LIN {X 0,Y 227.871,Z 414.724,A -85,B 0,C 180,E1 -20018.086,E2 -20018.086} C_VEL
LIN {X 0,Y 228.23,Z 417.25,A -85,B 0,C 180,E1 -20022.645,E2 -20022.645} C_VEL
LIN {X 0,Y 228.444,Z 418.737,A -85,B 0,C 180,E1 -20025.039,E2 -20025.039} C_VEL
LIN {X 0,Y 228.671,Z 421.522,A -85,B 0,C 180,E1 -20029.238,E2 -20029.238} C_VEL
LIN {X 0,Y 228.672,Z 421.631,A -85,B 0,C 180,E1 -20029.384,E2 -20029.384} C_VEL
LIN {X 0,Y 229.708,Z 424.715,A -85,B 0,C 180,E1 -20029.753,E2 -20029.753} C_VEL
LIN {X 0,Y 231.122,Z 427.161,A -85,B 0,C 180,E1 -20030.178,E2 -20030.178} C_VEL
LIN {X 0,Y 235.965,Z 438.096,A -85,B 0,C 180,E1 -20031.887,E2 -20031.887} C_VEL
LIN {X 0,Y 239.913,Z 449.78,A -85,B 0,C 180,E1 -20033.668,E2 -20033.668} C_VEL
LIN {X 0,Y 243.067,Z 462.472,A -85,B 0,C 180,E1 -20035.659,E2 -20035.659} C_VEL
LIN {X 0,Y 244.778,Z 473.661,A -85,B 0,C 180,E1 -20037.501,E2 -20037.501} C_VEL
LIN {X 0,Y 245.596,Z 484.037,A -85,B 0,C 180,E1 -20039.347,E2 -20039.347} C_VEL
LIN {X 0,Y 242.616,Z 495.451,A -85,B 0,C 180,E1 -20041.211,E2 -20041.211} C_VEL
LIN {X 0,Y 239.291,Z 506.287,A -85,B 0,C 180,E1 -20043.392,E2 -20043.392} C_VEL
LIN {X 0,Y 236.26,Z 516.038,A -85,B 0,C 180,E1 -20045.857,E2 -20045.857} C_VEL
LIN {X 0,Y 233.502,Z 524.128,A -85,B 0,C 180,E1 -20048.364,E2 -20048.364} C_VEL
LIN {X 0,Y 231.017,Z 531.87,A -85,B 0,C 180,E1 -20051.372,E2 -20051.372} C_VEL
LIN {X 0,Y 229.237,Z 537.277,A -85,B 0,C 180,E1 -20053.983,E2 -20053.983} C_VEL
LIN {X 0,Y 227.771,Z 541.724,A -85,B 0,C 180,E1 -20056.62,E2 -20056.62} C_VEL
LIN {X 0,Y 226.783,Z 545.213,A -85,B 0,C 180,E1 -20059.284,E2 -20059.284} C_VEL
LIN {X 0,Y 226,Z 548.612,A -85,B 0,C 180,E1 -20062.855,E2 -20062.855} C_VEL
LIN {X 0,Y 225.629,Z 550.629,A -85,B 0,C 180,E1 -20066.428,E2 -20066.428} C_VEL
LIN {X 0,Y 225.637,Z 551.315,A -85,B 0,C 180,E1 -20070,E2 -20070} C_VEL
LIN {X 0,Y 225.629,Z 550.682,A -85,B 0,C 180,E1 -20073.572,E2 -20073.572} C_VEL
LIN {X 0,Y 225.998,Z 548.713,A -85,B 0,C 180,E1 -20077.146,E2 -20077.146} C_VEL
LIN {X 0,Y 226.763,Z 545.363,A -85,B 0,C 180,E1 -20080.717,E2 -20080.717} C_VEL
LIN {X 0,Y 228.133,Z 540.531,A -85,B 0,C 180,E1 -20084.268,E2 -20084.268} C_VEL
LIN {X 0,Y 230.402,Z 534.059,A -85,B 0,C 180,E1 -20087.76,E2 -20087.76} C_VEL
LIN {X 0,Y 232.445,Z 527.554,A -85,B 0,C 180,E1 -20090.519,E2 -20090.519} C_VEL
LIN {X 0,Y 235.212,Z 519.304,A -85,B 0,C 180,E1 -20093.323,E2 -20093.323} C_VEL
LIN {X 0,Y 238.194,Z 510.234,A -85,B 0,C 180,E1 -20095.799,E2 -20095.799} C_VEL
LIN {X 0,Y 241.6,Z 499.245,A -85,B 0,C 180,E1 -20098.21,E2 -20098.21} C_VEL
LIN {X 0,Y 244.722,Z 487.841,A -85,B 0,C 180,E1 -20100.206,E2 -20100.206} C_VEL
LIN {X 0,Y 245.654,Z 482.869,A -85,B 0,C 180,E1 -20100.996,E2 -20100.996} C_VEL
LIN {X 0,Y 244.462,Z 470.906,A -85,B 0,C 180,E1 -20103.109,E2 -20103.109} C_VEL
LIN {X 0,Y 242.661,Z 460.374,A -85,B 0,C 180,E1 -20104.815,E2 -20104.815} C_VEL
LIN {X 0,Y 239.265,Z 447.447,A -85,B 0,C 180,E1 -20106.828,E2 -20106.828} C_VEL
LIN {X 0,Y 235.103,Z 435.976,A -85,B 0,C 180,E1 -20108.587,E2 -20108.587} C_VEL
LIN {X 0,Y 232.091,Z 429.289,A -85,B 0,C 180,E1 -20109.642,E2 -20109.642} C_VEL
LIN {X 0,Y 230.405,Z 425.764,A -85,B 0,C 180,E1 -20110.203,E2 -20110.203} C_VEL
LIN {X 0,Y 228.882,Z 422.633,A -85,B 0,C 180,E1 -20110.677,E2 -20110.677} C_VEL
LIN {X 0,Y 228.676,Z 421.578,A -85,B 0,C 180,E1 -20110.836,E2 -20110.836} C_VEL
LIN {X 0,Y 228.449,Z 418.795,A -85,B 0,C 180,E1 -20115.038,E2 -20115.038} C_VEL
LIN {X 0,Y 228.031,Z 415.991,A -85,B 0,C 180,E1 -20119.667,E2 -20119.667} C_VEL
LIN {X 0,Y 227.849,Z 414.733,A -85,B 0,C 180,E1 -20121.91,E2 -20121.91} C_VEL
LIN {X 0,Y 227.881,Z 414.724,A -85,B 0,C 180,E1 -20126.377,E2 -20126.377} C_VEL
LIN {X 0,Y 227.922,Z 414.716,A -85,B 0,C 180,E1 -20130.438,E2 -20130.438} C_VEL
LIN {X 0,Y 227.931,Z 414.719,A -85,B 0,C 180,E1 -20134.426,E2 -20134.426} C_VEL
LIN {X 0,Y 227.965,Z 414.714,A -85,B 0,C 180,E1 -20138.287,E2 -20138.287} C_VEL
LIN {X 0,Y 228.037,Z 414.705,A -85,B 0,C 180,E1 -20142.825,E2 -20142.825} C_VEL
LIN {X 0,Y 228.097,Z 414.698,A -85,B 0,C 180,E1 -20147.544,E2 -20147.544} C_VEL
LIN {X 0,Y 228.328,Z 414.666,A -85,B 0,C 180,E1 -20151.147,E2 -20151.147} C_VEL
LIN {X 0,Y 228.361,Z 414.665,A -85,B 0,C 180,E1 -20152.929,E2 -20152.929} C_VEL
LIN {X 0,Y 228.557,Z 414.639,A -85,B 0,C 180,E1 -20158.238,E2 -20158.238} C_VEL
LIN {X 0,Y 228.558,Z 414.641,A -85,B 0,C 180,E1 -20161.762,E2 -20161.762} C_VEL
LIN {X 0,Y 228.361,Z 414.665,A -85,B 0,C 180,E1 -20167.071,E2 -20167.071} C_VEL
LIN {X 0,Y 228.174,Z 414.687,A -85,B 0,C 180,E1 -20170.65,E2 -20170.65} C_VEL
LIN {X 0,Y 228.06,Z 414.704,A -85,B 0,C 180,E1 -20176.102,E2 -20176.102} C_VEL
LIN {X 0,Y 227.945,Z 414.718,A -85,B 0,C 180,E1 -20179.825,E2 -20179.825} C_VEL
LIN {X 0,Y 227.916,Z 414.713,A -85,B 0,C 180,E1 -20183.632,E2 -20183.632} C_VEL
LIN {X 0,Y 227.888,Z 414.718,A -85,B 0,C 180,E1 -20187.555,E2 -20187.555} C_VEL
LIN {X 0,Y 227.875,Z 414.726,A -85,B 0,C 180,E1 -20191.621,E2 -20191.621} C_VEL
LIN {X 0,Y 227.892,Z 414.725,A -85,B 0,C 180,E1 -20193.718,E2 -20193.718} C_VEL
LIN {X 0,Y 228.131,Z 416.119,A -85,B 0,C 180,E1 -20196.776,E2 -20196.776} C_VEL
LIN {X 0,Y 228.439,Z 418.282,A -85,B 0,C 180,E1 -20200.246,E2 -20200.246} C_VEL
LIN {X 0,Y 228.732,Z 419.796,A -85,B 0,C 180,E1 -20202.53,E2 -20202.53} C_VEL
LIN {X 0,Y 228.948,Z 421.571,A -85,B 0,C 180,E1 -20205.087,E2 -20205.087} C_VEL
LIN {X 0,Y 229.149,Z 424.277,A -85,B 0,C 180,E1 -20208.712,E2 -20208.712} C_VEL
LIN {X 0,Y 229.127,Z 424.775,A -85,B 0,C 180,E1 -20209.344,E2 -20209.344} C_VEL
LIN {X 0,Y 230.212,Z 428.044,A -85,B 0,C 180,E1 -20209.748,E2 -20209.748} C_VEL
LIN {X 0,Y 231.469,Z 430.266,A -85,B 0,C 180,E1 -20210.122,E2 -20210.122} C_VEL
LIN {X 0,Y 235.394,Z 439.747,A -85,B 0,C 180,E1 -20211.529,E2 -20211.529} C_VEL
LIN {X 0,Y 239.443,Z 452.197,A -85,B 0,C 180,E1 -20213.352,E2 -20213.352} C_VEL
LIN {X 0,Y 240.173,Z 457.38,A -85,B 0,C 180,E1 -20214.014,E2 -20214.014} C_VEL
LIN {X 0,Y 239.976,Z 462.788,A -85,B 0,C 180,E1 -20214.601,E2 -20214.601} C_VEL
LIN {X 0,Y 238.366,Z 473.596,A -85,B 0,C 180,E1 -20215.801,E2 -20215.801} C_VEL
LIN {X 0,Y 237.926,Z 478.732,A -85,B 0,C 180,E1 -20216.526,E2 -20216.526} C_VEL
LIN {X 0,Y 237.969,Z 480.365,A -85,B 0,C 180,E1 -20216.8,E2 -20216.8} C_VEL
LIN {X 0,Y 238.435,Z 490.141,A -85,B 0,C 180,E1 -20218.626,E2 -20218.626} C_VEL
LIN {X 0,Y 235.967,Z 499.91,A -85,B 0,C 180,E1 -20220.32,E2 -20220.32} C_VEL
LIN {X 0,Y 232.489,Z 510.701,A -85,B 0,C 180,E1 -20222.548,E2 -20222.548} C_VEL
LIN {X 0,Y 229.263,Z 520.429,A -85,B 0,C 180,E1 -20225.07,E2 -20225.07} C_VEL
LIN {X 0,Y 226.424,Z 528.498,A -85,B 0,C 180,E1 -20227.652,E2 -20227.652} C_VEL
LIN {X 0,Y 224.105,Z 534.99,A -85,B 0,C 180,E1 -20230.187,E2 -20230.187} C_VEL
LIN {X 0,Y 222.033,Z 541.634,A -85,B 0,C 180,E1 -20233.448,E2 -20233.448} C_VEL
LIN {X 0,Y 220.123,Z 547.315,A -85,B 0,C 180,E1 -20237.085,E2 -20237.085} C_VEL
LIN {X 0,Y 219.076,Z 551.438,A -85,B 0,C 180,E1 -20240.77,E2 -20240.77} C_VEL
LIN {X 0,Y 218.567,Z 554.13,A -85,B 0,C 180,E1 -20244.464,E2 -20244.464} C_VEL
LIN {X 0,Y 218.467,Z 555.461,A -85,B 0,C 180,E1 -20248.156,E2 -20248.156} C_VEL
LIN {X 0,Y 218.532,Z 555.625,A -85,B 0,C 180,E1 -20250,E2 -20250} C_VEL
LIN {X 0,Y 218.449,Z 554.948,A -85,B 0,C 180,E1 -20253.689,E2 -20253.689} C_VEL
LIN {X 0,Y 218.758,Z 552.928,A -85,B 0,C 180,E1 -20257.383,E2 -20257.383} C_VEL
LIN {X 0,Y 219.552,Z 549.517,A -85,B 0,C 180,E1 -20261.073,E2 -20261.073} C_VEL
LIN {X 0,Y 220.952,Z 544.612,A -85,B 0,C 180,E1 -20264.742,E2 -20264.742} C_VEL
LIN {X 0,Y 222.567,Z 539.883,A -85,B 0,C 180,E1 -20267.456,E2 -20267.456} C_VEL
LIN {X 0,Y 224.851,Z 533.028,A -85,B 0,C 180,E1 -20270.587,E2 -20270.587} C_VEL
LIN {X 0,Y 227.79,Z 524.519,A -85,B 0,C 180,E1 -20273.646,E2 -20273.646} C_VEL
LIN {X 0,Y 230.836,Z 515.642,A -85,B 0,C 180,E1 -20276.197,E2 -20276.197} C_VEL
LIN {X 0,Y 234.347,Z 504.889,A -85,B 0,C 180,E1 -20278.675,E2 -20278.675} C_VEL
LIN {X 0,Y 237.768,Z 493.13,A -85,B 0,C 180,E1 -20280.839,E2 -20280.839} C_VEL
LIN {X 0,Y 238.393,Z 489.802,A -85,B 0,C 180,E1 -20281.396,E2 -20281.396} C_VEL
LIN {X 0,Y 237.762,Z 478.712,A -85,B 0,C 180,E1 -20283.448,E2 -20283.448} C_VEL
LIN {X 0,Y 236.133,Z 466.35,A -85,B 0,C 180,E1 -20285.536,E2 -20285.536} C_VEL
LIN {X 0,Y 233.476,Z 454.446,A -85,B 0,C 180,E1 -20287.445,E2 -20287.445} C_VEL
LIN {X 0,Y 229.625,Z 442.08,A -85,B 0,C 180,E1 -20289.376,E2 -20289.376} C_VEL
LIN {X 0,Y 226.084,Z 433.454,A -85,B 0,C 180,E1 -20290.753,E2 -20290.753} C_VEL
LIN {X 0,Y 223.799,Z 428.789,A -85,B 0,C 180,E1 -20291.548,E2 -20291.548} C_VEL
LIN {X 0,Y 222.268,Z 425.689,A -85,B 0,C 180,E1 -20292.054,E2 -20292.054} C_VEL
LIN {X 0,Y 222.084,Z 424.67,A -85,B 0,C 180,E1 -20292.188,E2 -20292.188} C_VEL
LIN {X 0,Y 221.733,Z 421.441,A -85,B 0,C 180,E1 -20296.803,E2 -20296.803} C_VEL
LIN {X 0,Y 221.37,Z 419.006,A -85,B 0,C 180,E1 -20300.583,E2 -20300.583} C_VEL
LIN {X 0,Y 220.945,Z 416.375,A -85,B 0,C 180,E1 -20305.071,E2 -20305.071} C_VEL
LIN {X 0,Y 220.824,Z 415.606,A -85,B 0,C 180,E1 -20307.245,E2 -20307.245} C_VEL
LIN {X 0,Y 220.827,Z 415.604,A -85,B 0,C 180,E1 -20311.485,E2 -20311.485} C_VEL
LIN {X 0,Y 220.863,Z 415.599,A -85,B 0,C 180,E1 -20315.565,E2 -20315.565} C_VEL
LIN {X 0,Y 220.886,Z 415.596,A -85,B 0,C 180,E1 -20319.513,E2 -20319.513} C_VEL
LIN {X 0,Y 221.018,Z 415.579,A -85,B 0,C 180,E1 -20323.37,E2 -20323.37} C_VEL
LIN {X 0,Y 221.118,Z 415.561,A -85,B 0,C 180,E1 -20329.006,E2 -20329.006} C_VEL
LIN {X 0,Y 221.313,Z 415.535,A -85,B 0,C 180,E1 -20332.702,E2 -20332.702} C_VEL
LIN {X 0,Y 221.515,Z 415.517,A -85,B 0,C 180,E1 -20338.182,E2 -20338.182} C_VEL
LIN {X 0,Y 221.514,Z 415.517,A -85,B 0,C 180,E1 -20341.818,E2 -20341.818} C_VEL
LIN {X 0,Y 221.313,Z 415.543,A -85,B 0,C 180,E1 -20347.298,E2 -20347.298} C_VEL
LIN {X 0,Y 221.118,Z 415.566,A -85,B 0,C 180,E1 -20350.994,E2 -20350.994} C_VEL
LIN {X 0,Y 221.018,Z 415.574,A -85,B 0,C 180,E1 -20356.63,E2 -20356.63} C_VEL
LIN {X 0,Y 220.894,Z 415.595,A -85,B 0,C 180,E1 -20360.486,E2 -20360.486} C_VEL
LIN {X 0,Y 220.869,Z 415.598,A -85,B 0,C 180,E1 -20364.435,E2 -20364.435} C_VEL
LIN {X 0,Y 220.828,Z 415.603,A -85,B 0,C 180,E1 -20368.515,E2 -20368.515} C_VEL
LIN {X 0,Y 220.824,Z 415.604,A -85,B 0,C 180,E1 -20372.755,E2 -20372.755} C_VEL
LIN {X 0,Y 220.839,Z 415.603,A -85,B 0,C 180,E1 -20377.288,E2 -20377.288} C_VEL
LIN {X 0,Y 221.18,Z 418.058,A -85,B 0,C 180,E1 -20381.857,E2 -20381.857} C_VEL
LIN {X 0,Y 221.472,Z 420.385,A -85,B 0,C 180,E1 -20385.723,E2 -20385.723} C_VEL
LIN {X 0,Y 221.635,Z 421.75,A -85,B 0,C 180,E1 -20387.805,E2 -20387.805} C_VEL
LIN {X 0,Y 222.739,Z 424.806,A -85,B 0,C 180,E1 -20388.217,E2 -20388.217} C_VEL
LIN {X 0,Y 224.207,Z 427.147,A -85,B 0,C 180,E1 -20388.68,E2 -20388.68} C_VEL
LIN {X 0,Y 229.392,Z 438.499,A -85,B 0,C 180,E1 -20390.611,E2 -20390.611} C_VEL
LIN {X 0,Y 233.08,Z 448.969,A -85,B 0,C 180,E1 -20392.328,E2 -20392.328} C_VEL
LIN {X 0,Y 236.412,Z 461.889,A -85,B 0,C 180,E1 -20394.462,E2 -20394.462} C_VEL
LIN {X 0,Y 238.314,Z 473.741,A -85,B 0,C 180,E1 -20396.505,E2 -20396.505} C_VEL
LIN {X 0,Y 239.179,Z 484.183,A -85,B 0,C 180,E1 -20398.445,E2 -20398.445} C_VEL
LIN {X 0,Y 238.474,Z 488.194,A -85,B 0,C 180,E1 -20399.11,E2 -20399.11} C_VEL
LIN {X 0,Y 235.433,Z 498.727,A -85,B 0,C 180,E1 -20400.982,E2 -20400.982} C_VEL
LIN {X 0,Y 232.395,Z 508.137,A -85,B 0,C 180,E1 -20403.024,E2 -20403.024} C_VEL
LIN {X 0,Y 229.244,Z 517.592,A -85,B 0,C 180,E1 -20405.552,E2 -20405.552} C_VEL
LIN {X 0,Y 226.026,Z 526.63,A -85,B 0,C 180,E1 -20408.58,E2 -20408.58} C_VEL
LIN {X 0,Y 223.66,Z 533.87,A -85,B 0,C 180,E1 -20411.686,E2 -20411.686} C_VEL
LIN {X 0,Y 221.248,Z 540.395,A -85,B 0,C 180,E1 -20415.279,E2 -20415.279} C_VEL
LIN {X 0,Y 219.772,Z 545.283,A -85,B 0,C 180,E1 -20418.938,E2 -20418.938} C_VEL
LIN {X 0,Y 218.943,Z 548.682,A -85,B 0,C 180,E1 -20422.623,E2 -20422.623} C_VEL
LIN {X 0,Y 218.534,Z 550.698,A -85,B 0,C 180,E1 -20426.312,E2 -20426.312} C_VEL
LIN {X 0,Y 218.537,Z 551.384,A -85,B 0,C 180,E1 -20430,E2 -20430} C_VEL
LIN {X 0,Y 218.534,Z 550.751,A -85,B 0,C 180,E1 -20433.688,E2 -20433.688} C_VEL
LIN {X 0,Y 218.941,Z 548.781,A -85,B 0,C 180,E1 -20437.377,E2 -20437.377} C_VEL
LIN {X 0,Y 219.75,Z 545.431,A -85,B 0,C 180,E1 -20441.063,E2 -20441.063} C_VEL
LIN {X 0,Y 221.225,Z 540.599,A -85,B 0,C 180,E1 -20444.723,E2 -20444.723} C_VEL
LIN {X 0,Y 222.978,Z 535.932,A -85,B 0,C 180,E1 -20447.423,E2 -20447.423} C_VEL
LIN {X 0,Y 225.301,Z 528.928,A -85,B 0,C 180,E1 -20450.639,E2 -20450.639} C_VEL
LIN {X 0,Y 228.203,Z 520.722,A -85,B 0,C 180,E1 -20453.601,E2 -20453.601} C_VEL
LIN {X 0,Y 231.227,Z 511.925,A -85,B 0,C 180,E1 -20456.15,E2 -20456.15} C_VEL
LIN {X 0,Y 234.73,Z 501.263,A -85,B 0,C 180,E1 -20458.624,E2 -20458.624} C_VEL
LIN {X 0,Y 238.108,Z 489.742,A -85,B 0,C 180,E1 -20460.762,E2 -20460.762} C_VEL
LIN {X 0,Y 239.256,Z 484.688,A -85,B 0,C 180,E1 -20461.585,E2 -20461.585} C_VEL
LIN {X 0,Y 238.265,Z 473.172,A -85,B 0,C 180,E1 -20463.735,E2 -20463.735} C_VEL
LIN {X 0,Y 236.669,Z 462.938,A -85,B 0,C 180,E1 -20465.5,E2 -20465.5} C_VEL
LIN {X 0,Y 233.693,Z 450.793,A -85,B 0,C 180,E1 -20467.514,E2 -20467.514} C_VEL
LIN {X 0,Y 229.547,Z 438.758,A -85,B 0,C 180,E1 -20469.491,E2 -20469.491} C_VEL
LIN {X 0,Y 225.551,Z 430.034,A -85,B 0,C 180,E1 -20470.988,E2 -20470.988} C_VEL
LIN {X 0,Y 223.627,Z 426.043,A -85,B 0,C 180,E1 -20471.676,E2 -20471.676} C_VEL
LIN {X 0,Y 222.021,Z 423.296,A -85,B 0,C 180,E1 -20472.186,E2 -20472.186} C_VEL
LIN {X 0,Y 221.616,Z 421.7,A -85,B 0,C 180,E1 -20472.386,E2 -20472.386} C_VEL
LIN {X 0,Y 221.263,Z 418.872,A -85,B 0,C 180,E1 -20476.933,E2 -20476.933} C_VEL
LIN {X 0,Y 221,Z 416.838,A -85,B 0,C 180,E1 -20480.504,E2 -20480.504} C_VEL
LIN {X 0,Y 220.826,Z 415.615,A -85,B 0,C 180,E1 -20482.793,E2 -20482.793} C_VEL
LIN {X 0,Y 220.82,Z 415.604,A -85,B 0,C 180,E1 -20487.244,E2 -20487.244} C_VEL
LIN {X 0,Y 220.839,Z 415.602,A -85,B 0,C 180,E1 -20491.487,E2 -20491.487} C_VEL
LIN {X 0,Y 220.87,Z 415.595,A -85,B 0,C 180,E1 -20495.565,E2 -20495.565} C_VEL
LIN {X 0,Y 220.895,Z 415.588,A -85,B 0,C 180,E1 -20499.514,E2 -20499.514} C_VEL
LIN {X 0,Y 221.019,Z 415.58,A -85,B 0,C 180,E1 -20503.37,E2 -20503.37} C_VEL
LIN {X 0,Y 221.12,Z 415.566,A -85,B 0,C 180,E1 -20509.006,E2 -20509.006} C_VEL
LIN {X 0,Y 221.314,Z 415.542,A -85,B 0,C 180,E1 -20512.702,E2 -20512.702} C_VEL
LIN {X 0,Y 221.515,Z 415.516,A -85,B 0,C 180,E1 -20518.182,E2 -20518.182} C_VEL
LIN {X 0,Y 221.516,Z 415.518,A -85,B 0,C 180,E1 -20521.818,E2 -20521.818} C_VEL
LIN {X 0,Y 221.314,Z 415.542,A -85,B 0,C 180,E1 -20527.297,E2 -20527.297} C_VEL
LIN {X 0,Y 221.119,Z 415.566,A -85,B 0,C 180,E1 -20530.994,E2 -20530.994} C_VEL
LIN {X 0,Y 221.019,Z 415.578,A -85,B 0,C 180,E1 -20536.629,E2 -20536.629} C_VEL
LIN {X 0,Y 220.895,Z 415.595,A -85,B 0,C 180,E1 -20540.486,E2 -20540.486} C_VEL
LIN {X 0,Y 220.869,Z 415.591,A -85,B 0,C 180,E1 -20544.435,E2 -20544.435} C_VEL
LIN {X 0,Y 220.839,Z 415.602,A -85,B 0,C 180,E1 -20548.513,E2 -20548.513} C_VEL
LIN {X 0,Y 220.826,Z 415.604,A -85,B 0,C 180,E1 -20552.754,E2 -20552.754} C_VEL
LIN {X 0,Y 220.954,Z 416.433,A -85,B 0,C 180,E1 -20554.927,E2 -20554.927} C_VEL
LIN {X 0,Y 221.378,Z 419.059,A -85,B 0,C 180,E1 -20559.415,E2 -20559.415} C_VEL
LIN {X 0,Y 221.756,Z 421.493,A -85,B 0,C 180,E1 -20563.203,E2 -20563.203} C_VEL
LIN {X 0,Y 222.158,Z 424.853,A -85,B 0,C 180,E1 -20567.808,E2 -20567.808} C_VEL
LIN {X 0,Y 223.3,Z 428.018,A -85,B 0,C 180,E1 -20568.231,E2 -20568.231} C_VEL
LIN {X 0,Y 224.65,Z 430.332,A -85,B 0,C 180,E1 -20568.661,E2 -20568.661} C_VEL
LIN {X 0,Y 229.373,Z 441.097,A -85,B 0,C 180,E1 -20570.434,E2 -20570.434} C_VEL
LIN {X 0,Y 233.591,Z 454.451,A -85,B 0,C 180,E1 -20572.519,E2 -20572.519} C_VEL
LIN {X 0,Y 235.977,Z 465.2,A -85,B 0,C 180,E1 -20574.231,E2 -20574.231} C_VEL
LIN {X 0,Y 237.489,Z 475.583,A -85,B 0,C 180,E1 -20575.956,E2 -20575.956} C_VEL
LIN {X 0,Y 237.969,Z 480.365,A -85,B 0,C 180,E1 -20576.8,E2 -20576.8} C_VEL
LIN {X 0,Y 237.788,Z 483.651,A -85,B 0,C 180,E1 -20577.331,E2 -20577.331} C_VEL
LIN {X 0,Y 236.364,Z 488.667,A -85,B 0,C 180,E1 -20578.031,E2 -20578.031} C_VEL
LIN {X 0,Y 234.087,Z 493.547,A -85,B 0,C 180,E1 -20578.67,E2 -20578.67} C_VEL
LIN {X 0,Y 229.005,Z 503.067,A -85,B 0,C 180,E1 -20580.09,E2 -20580.09} C_VEL
LIN {X 0,Y 227.778,Z 506.04,A -85,B 0,C 180,E1 -20580.685,E2 -20580.685} C_VEL
LIN {X 0,Y 224.427,Z 515.73,A -85,B 0,C 180,E1 -20582.995,E2 -20582.995} C_VEL
LIN {X 0,Y 221.297,Z 524.581,A -85,B 0,C 180,E1 -20585.615,E2 -20585.615} C_VEL
LIN {X 0,Y 218.145,Z 533.064,A -85,B 0,C 180,E1 -20588.749,E2 -20588.749} C_VEL
LIN {X 0,Y 215.743,Z 539.901,A -85,B 0,C 180,E1 -20591.972,E2 -20591.972} C_VEL
LIN {X 0,Y 214.077,Z 544.611,A -85,B 0,C 180,E1 -20594.773,E2 -20594.773} C_VEL
LIN {X 0,Y 212.546,Z 549.494,A -85,B 0,C 180,E1 -20598.557,E2 -20598.557} C_VEL
LIN {X 0,Y 211.667,Z 552.888,A -85,B 0,C 180,E1 -20602.368,E2 -20602.368} C_VEL
LIN {X 0,Y 211.349,Z 554.895,A -85,B 0,C 180,E1 -20606.186,E2 -20606.186} C_VEL
LIN {X 0,Y 211.434,Z 555.556,A -85,B 0,C 180,E1 -20610,E2 -20610} C_VEL
LIN {X 0,Y 211.354,Z 554.878,A -85,B 0,C 180,E1 -20613.813,E2 -20613.813} C_VEL
LIN {X 0,Y 211.685,Z 552.858,A -85,B 0,C 180,E1 -20617.631,E2 -20617.631} C_VEL
LIN {X 0,Y 212.534,Z 549.446,A -85,B 0,C 180,E1 -20621.444,E2 -20621.444} C_VEL
LIN {X 0,Y 214.075,Z 544.541,A -85,B 0,C 180,E1 -20625.226,E2 -20625.226} C_VEL
LIN {X 0,Y 216.442,Z 538,A -85,B 0,C 180,E1 -20628.948,E2 -20628.948} C_VEL
LIN {X 0,Y 218.959,Z 530.72,A -85,B 0,C 180,E1 -20632.157,E2 -20632.157} C_VEL
LIN {X 0,Y 222.296,Z 521.703,A -85,B 0,C 180,E1 -20635.265,E2 -20635.265} C_VEL
LIN {X 0,Y 225.578,Z 512.242,A -85,B 0,C 180,E1 -20637.861,E2 -20637.861} C_VEL
LIN {X 0,Y 229.095,Z 501.769,A -85,B 0,C 180,E1 -20640.155,E2 -20640.155} C_VEL
LIN {X 0,Y 231.991,Z 491.683,A -85,B 0,C 180,E1 -20641.979,E2 -20641.979} C_VEL
LIN {X 0,Y 231.584,Z 481.339,A -85,B 0,C 180,E1 -20644.008,E2 -20644.008} C_VEL
LIN {X 0,Y 230.147,Z 468.823,A -85,B 0,C 180,E1 -20646.257,E2 -20646.257} C_VEL
LIN {X 0,Y 227.602,Z 456.606,A -85,B 0,C 180,E1 -20648.335,E2 -20648.335} C_VEL
LIN {X 0,Y 223.683,Z 443.741,A -85,B 0,C 180,E1 -20650.484,E2 -20650.484} C_VEL
LIN {X 0,Y 219.427,Z 433.674,A -85,B 0,C 180,E1 -20652.246,E2 -20652.246} C_VEL
LIN {X 0,Y 217.641,Z 429.973,A -85,B 0,C 180,E1 -20652.928,E2 -20652.928} C_VEL
LIN {X 0,Y 215.472,Z 426.425,A -85,B 0,C 180,E1 -20653.661,E2 -20653.661} C_VEL
LIN {X 0,Y 214.984,Z 424.57,A -85,B 0,C 180,E1 -20653.951,E2 -20653.951} C_VEL
LIN {X 0,Y 214.756,Z 422.805,A -85,B 0,C 180,E1 -20656.588,E2 -20656.588} C_VEL
LIN {X 0,Y 214.538,Z 421.232,A -85,B 0,C 180,E1 -20659.067,E2 -20659.067} C_VEL
LIN {X 0,Y 214.081,Z 418.468,A -85,B 0,C 180,E1 -20663.778,E2 -20663.778} C_VEL
LIN {X 0,Y 213.903,Z 417.245,A -85,B 0,C 180,E1 -20666.044,E2 -20666.044} C_VEL
LIN {X 0,Y 213.782,Z 416.484,A -85,B 0,C 180,E1 -20668.731,E2 -20668.731} C_VEL
LIN {X 0,Y 213.827,Z 416.476,A -85,B 0,C 180,E1 -20672.603,E2 -20672.603} C_VEL
LIN {X 0,Y 213.82,Z 416.476,A -85,B 0,C 180,E1 -20676.974,E2 -20676.974} C_VEL
LIN {X 0,Y 213.945,Z 416.457,A -85,B 0,C 180,E1 -20682.804,E2 -20682.804} C_VEL
LIN {X 0,Y 213.982,Z 416.455,A -85,B 0,C 180,E1 -20686.709,E2 -20686.709} C_VEL
LIN {X 0,Y 214.198,Z 416.43,A -85,B 0,C 180,E1 -20690.558,E2 -20690.558} C_VEL
LIN {X 0,Y 214.25,Z 416.415,A -85,B 0,C 180,E1 -20692.461,E2 -20692.461} C_VEL
LIN {X 0,Y 214.448,Z 416.397,A -85,B 0,C 180,E1 -20698.122,E2 -20698.122} C_VEL
LIN {X 0,Y 214.556,Z 416.383,A -85,B 0,C 180,E1 -20700,E2 -20700} C_VEL
LIN {X 0,Y 214.447,Z 416.397,A -85,B 0,C 180,E1 -20701.878,E2 -20701.878} C_VEL
LIN {X 0,Y 214.25,Z 416.423,A -85,B 0,C 180,E1 -20707.54,E2 -20707.54} C_VEL
LIN {X 0,Y 214.049,Z 416.448,A -85,B 0,C 180,E1 -20711.362,E2 -20711.362} C_VEL
LIN {X 0,Y 213.936,Z 416.462,A -85,B 0,C 180,E1 -20715.237,E2 -20715.237} C_VEL
LIN {X 0,Y 213.842,Z 416.474,A -85,B 0,C 180,E1 -20719.187,E2 -20719.187} C_VEL
LIN {X 0,Y 213.849,Z 416.472,A -85,B 0,C 180,E1 -20723.227,E2 -20723.227} C_VEL
LIN {X 0,Y 213.83,Z 416.474,A -85,B 0,C 180,E1 -20727.45,E2 -20727.45} C_VEL
LIN {X 0,Y 213.771,Z 416.483,A -85,B 0,C 180,E1 -20731.737,E2 -20731.737} C_VEL
LIN {X 0,Y 213.754,Z 416.486,A -85,B 0,C 180,E1 -20736.287,E2 -20736.287} C_VEL
LIN {X 0,Y 214.126,Z 418.891,A -85,B 0,C 180,E1 -20741.029,E2 -20741.029} C_VEL
LIN {X 0,Y 214.488,Z 421.794,A -85,B 0,C 180,E1 -20746.045,E2 -20746.045} C_VEL
LIN {X 0,Y 215.593,Z 424.821,A -85,B 0,C 180,E1 -20746.491,E2 -20746.491} C_VEL
LIN {X 0,Y 217.434,Z 427.586,A -85,B 0,C 180,E1 -20747.115,E2 -20747.115} C_VEL
LIN {X 0,Y 221.729,Z 436.437,A -85,B 0,C 180,E1 -20748.785,E2 -20748.785} C_VEL
LIN {X 0,Y 225.509,Z 445.84,A -85,B 0,C 180,E1 -20750.474,E2 -20750.474} C_VEL
LIN {X 0,Y 228.574,Z 456.158,A -85,B 0,C 180,E1 -20752.277,E2 -20752.277} C_VEL
LIN {X 0,Y 231.09,Z 467.811,A -85,B 0,C 180,E1 -20754.355,E2 -20754.355} C_VEL
LIN {X 0,Y 232.387,Z 478.742,A -85,B 0,C 180,E1 -20756.379,E2 -20756.379} C_VEL
LIN {X 0,Y 232.749,Z 486.796,A -85,B 0,C 180,E1 -20757.972,E2 -20757.972} C_VEL
LIN {X 0,Y 229.599,Z 497.731,A -85,B 0,C 180,E1 -20759.918,E2 -20759.918} C_VEL
LIN {X 0,Y 226.059,Z 508.209,A -85,B 0,C 180,E1 -20762.203,E2 -20762.203} C_VEL
LIN {X 0,Y 222.795,Z 517.664,A -85,B 0,C 180,E1 -20764.795,E2 -20764.795} C_VEL
LIN {X 0,Y 219.417,Z 526.681,A -85,B 0,C 180,E1 -20767.892,E2 -20767.892} C_VEL
LIN {X 0,Y 216.865,Z 533.941,A -85,B 0,C 180,E1 -20771.091,E2 -20771.091} C_VEL
LIN {X 0,Y 214.947,Z 539.026,A -85,B 0,C 180,E1 -20773.864,E2 -20773.864} C_VEL
LIN {X 0,Y 213.152,Z 544.292,A -85,B 0,C 180,E1 -20777.625,E2 -20777.625} C_VEL
LIN {X 0,Y 212.259,Z 547.231,A -85,B 0,C 180,E1 -20780.471,E2 -20780.471} C_VEL
LIN {X 0,Y 211.638,Z 549.928,A -85,B 0,C 180,E1 -20784.283,E2 -20784.283} C_VEL
LIN {X 0,Y 211.401,Z 551.275,A -85,B 0,C 180,E1 -20788.095,E2 -20788.095} C_VEL
LIN {X 0,Y 211.439,Z 551.452,A -85,B 0,C 180,E1 -20790,E2 -20790} C_VEL
LIN {X 0,Y 211.442,Z 550.819,A -85,B 0,C 180,E1 -20793.812,E2 -20793.812} C_VEL
LIN {X 0,Y 211.88,Z 548.85,A -85,B 0,C 180,E1 -20797.625,E2 -20797.625} C_VEL
LIN {X 0,Y 212.763,Z 545.5,A -85,B 0,C 180,E1 -20801.431,E2 -20801.431} C_VEL
LIN {X 0,Y 214.335,Z 540.667,A -85,B 0,C 180,E1 -20805.208,E2 -20805.208} C_VEL
LIN {X 0,Y 216.185,Z 535.999,A -85,B 0,C 180,E1 -20807.989,E2 -20807.989} C_VEL
LIN {X 0,Y 218.484,Z 529.442,A -85,B 0,C 180,E1 -20811.116,E2 -20811.116} C_VEL
LIN {X 0,Y 221.207,Z 522.138,A -85,B 0,C 180,E1 -20813.897,E2 -20813.897} C_VEL
LIN {X 0,Y 224.3,Z 513.613,A -85,B 0,C 180,E1 -20816.519,E2 -20816.519} C_VEL
LIN {X 0,Y 227.895,Z 503.277,A -85,B 0,C 180,E1 -20819.059,E2 -20819.059} C_VEL
LIN {X 0,Y 231.51,Z 491.597,A -85,B 0,C 180,E1 -20821.349,E2 -20821.349} C_VEL
LIN {X 0,Y 232.879,Z 485.901,A -85,B 0,C 180,E1 -20822.327,E2 -20822.327} C_VEL
LIN {X 0,Y 232.09,Z 475.414,A -85,B 0,C 180,E1 -20824.396,E2 -20824.396} C_VEL
LIN {X 0,Y 230.858,Z 466.363,A -85,B 0,C 180,E1 -20826.056,E2 -20826.056} C_VEL
LIN {X 0,Y 228.116,Z 454.111,A -85,B 0,C 180,E1 -20828.22,E2 -20828.22} C_VEL
LIN {X 0,Y 224.021,Z 441.753,A -85,B 0,C 180,E1 -20830.395,E2 -20830.395} C_VEL
LIN {X 0,Y 219.21,Z 430.931,A -85,B 0,C 180,E1 -20832.388,E2 -20832.388} C_VEL
LIN {X 0,Y 217.298,Z 427.201,A -85,B 0,C 180,E1 -20833.11,E2 -20833.11} C_VEL
LIN {X 0,Y 215.077,Z 423.811,A -85,B 0,C 180,E1 -20833.862,E2 -20833.862} C_VEL
LIN {X 0,Y 214.505,Z 421.764,A -85,B 0,C 180,E1 -20834.161,E2 -20834.161} C_VEL
LIN {X 0,Y 214.124,Z 418.969,A -85,B 0,C 180,E1 -20839.018,E2 -20839.018} C_VEL
LIN {X 0,Y 213.746,Z 416.533,A -85,B 0,C 180,E1 -20843.712,E2 -20843.712} C_VEL
LIN {X 0,Y 213.797,Z 416.478,A -85,B 0,C 180,E1 -20848.725,E2 -20848.725} C_VEL
LIN {X 0,Y 213.828,Z 416.475,A -85,B 0,C 180,E1 -20852.603,E2 -20852.603} C_VEL
LIN {X 0,Y 213.855,Z 416.468,A -85,B 0,C 180,E1 -20856.953,E2 -20856.953} C_VEL
LIN {X 0,Y 213.947,Z 416.46,A -85,B 0,C 180,E1 -20862.804,E2 -20862.804} C_VEL
LIN {X 0,Y 213.984,Z 416.454,A -85,B 0,C 180,E1 -20866.708,E2 -20866.708} C_VEL
LIN {X 0,Y 214.199,Z 416.428,A -85,B 0,C 180,E1 -20870.558,E2 -20870.558} C_VEL
LIN {X 0,Y 214.251,Z 416.423,A -85,B 0,C 180,E1 -20872.46,E2 -20872.46} C_VEL
LIN {X 0,Y 214.448,Z 416.396,A -85,B 0,C 180,E1 -20878.122,E2 -20878.122} C_VEL
LIN {X 0,Y 214.553,Z 416.385,A -85,B 0,C 180,E1 -20880,E2 -20880} C_VEL
LIN {X 0,Y 214.449,Z 416.399,A -85,B 0,C 180,E1 -20881.878,E2 -20881.878} C_VEL
LIN {X 0,Y 214.251,Z 416.422,A -85,B 0,C 180,E1 -20887.539,E2 -20887.539} C_VEL
LIN {X 0,Y 214.05,Z 416.449,A -85,B 0,C 180,E1 -20891.361,E2 -20891.361} C_VEL
LIN {X 0,Y 213.936,Z 416.461,A -85,B 0,C 180,E1 -20895.237,E2 -20895.237} C_VEL
LIN {X 0,Y 213.842,Z 416.472,A -85,B 0,C 180,E1 -20899.187,E2 -20899.187} C_VEL
LIN {X 0,Y 213.849,Z 416.466,A -85,B 0,C 180,E1 -20903.227,E2 -20903.227} C_VEL
LIN {X 0,Y 213.831,Z 416.468,A -85,B 0,C 180,E1 -20907.45,E2 -20907.45} C_VEL
LIN {X 0,Y 213.781,Z 416.481,A -85,B 0,C 180,E1 -20911.735,E2 -20911.735} C_VEL
LIN {X 0,Y 213.979,Z 417.75,A -85,B 0,C 180,E1 -20914.803,E2 -20914.803} C_VEL
LIN {X 0,Y 214.31,Z 419.855,A -85,B 0,C 180,E1 -20918.541,E2 -20918.541} C_VEL
LIN {X 0,Y 214.587,Z 421.399,A -85,B 0,C 180,E1 -20921.124,E2 -20921.124} C_VEL
LIN {X 0,Y 214.822,Z 423.219,A -85,B 0,C 180,E1 -20923.966,E2 -20923.966} C_VEL
LIN {X 0,Y 214.998,Z 424.658,A -85,B 0,C 180,E1 -20926.046,E2 -20926.046} C_VEL
LIN {X 0,Y 216.144,Z 427.81,A -85,B 0,C 180,E1 -20926.506,E2 -20926.506} C_VEL
LIN {X 0,Y 217.699,Z 430.009,A -85,B 0,C 180,E1 -20927.014,E2 -20927.014} C_VEL
LIN {X 0,Y 219.542,Z 433.856,A -85,B 0,C 180,E1 -20927.721,E2 -20927.721} C_VEL
LIN {X 0,Y 224.188,Z 444.925,A -85,B 0,C 180,E1 -20929.673,E2 -20929.673} C_VEL
LIN {X 0,Y 227.983,Z 457.776,A -85,B 0,C 180,E1 -20931.823,E2 -20931.823} C_VEL
LIN {X 0,Y 230.449,Z 470.213,A -85,B 0,C 180,E1 -20933.95,E2 -20933.95} C_VEL
LIN {X 0,Y 231.702,Z 482.333,A -85,B 0,C 180,E1 -20936.14,E2 -20936.14} C_VEL
LIN {X 0,Y 232.018,Z 491.868,A -85,B 0,C 180,E1 -20938.01,E2 -20938.01} C_VEL
LIN {X 0,Y 228.781,Z 503.046,A -85,B 0,C 180,E1 -20940.053,E2 -20940.053} C_VEL
LIN {X 0,Y 227.778,Z 506.04,A -85,B 0,C 180,E1 -20940.685,E2 -20940.685} C_VEL
LIN {X 0,Y 225.748,Z 510.354,A -85,B 0,C 180,E1 -20941.57,E2 -20941.57} C_VEL
LIN {X 0,Y 220.826,Z 517.084,A -85,B 0,C 180,E1 -20942.948,E2 -20942.948} C_VEL
LIN {X 0,Y 215.894,Z 523.327,A -85,B 0,C 180,E1 -20944.499,E2 -20944.499} C_VEL
LIN {X 0,Y 213.891,Z 526.864,A -85,B 0,C 180,E1 -20945.64,E2 -20945.64} C_VEL
LIN {X 0,Y 211.095,Z 534.079,A -85,B 0,C 180,E1 -20948.517,E2 -20948.517} C_VEL
LIN {X 0,Y 208.955,Z 539.833,A -85,B 0,C 180,E1 -20951.366,E2 -20951.366} C_VEL
LIN {X 0,Y 207.215,Z 544.543,A -85,B 0,C 180,E1 -20954.256,E2 -20954.256} C_VEL
LIN {X 0,Y 205.544,Z 549.425,A -85,B 0,C 180,E1 -20958.161,E2 -20958.161} C_VEL
LIN {X 0,Y 204.622,Z 552.82,A -85,B 0,C 180,E1 -20962.103,E2 -20962.103} C_VEL
LIN {X 0,Y 204.258,Z 554.879,A -85,B 0,C 180,E1 -20966.212,E2 -20966.212} C_VEL
LIN {X 0,Y 204.337,Z 555.487,A -85,B 0,C 180,E1 -20970,E2 -20970} C_VEL
LIN {X 0,Y 204.266,Z 554.809,A -85,B 0,C 180,E1 -20973.946,E2 -20973.946} C_VEL
LIN {X 0,Y 204.636,Z 552.789,A -85,B 0,C 180,E1 -20977.896,E2 -20977.896} C_VEL
LIN {X 0,Y 205.533,Z 549.376,A -85,B 0,C 180,E1 -20981.839,E2 -20981.839} C_VEL
LIN {X 0,Y 207.213,Z 544.471,A -85,B 0,C 180,E1 -20985.744,E2 -20985.744} C_VEL
LIN {X 0,Y 209.709,Z 537.93,A -85,B 0,C 180,E1 -20989.58,E2 -20989.58} C_VEL
LIN {X 0,Y 212.369,Z 530.649,A -85,B 0,C 180,E1 -20992.883,E2 -20992.883} C_VEL
LIN {X 0,Y 215.858,Z 521.631,A -85,B 0,C 180,E1 -20996.074,E2 -20996.074} C_VEL
LIN {X 0,Y 219.305,Z 512.171,A -85,B 0,C 180,E1 -20998.731,E2 -20998.731} C_VEL
LIN {X 0,Y 222.973,Z 501.697,A -85,B 0,C 180,E1 -21001.073,E2 -21001.073} C_VEL
LIN {X 0,Y 225.599,Z 492.811,A -85,B 0,C 180,E1 -21002.741,E2 -21002.741} C_VEL
LIN {X 0,Y 225.269,Z 482.516,A -85,B 0,C 180,E1 -21004.86,E2 -21004.86} C_VEL
LIN {X 0,Y 224.254,Z 472.094,A -85,B 0,C 180,E1 -21006.84,E2 -21006.84} C_VEL
LIN {X 0,Y 222.154,Z 460.644,A -85,B 0,C 180,E1 -21008.925,E2 -21008.925} C_VEL
LIN {X 0,Y 218.74,Z 448.174,A -85,B 0,C 180,E1 -21011.146,E2 -21011.146} C_VEL
LIN {X 0,Y 215.543,Z 440.077,A -85,B 0,C 180,E1 -21012.675,E2 -21012.675} C_VEL
LIN {X 0,Y 212.424,Z 433.586,A -85,B 0,C 180,E1 -21013.985,E2 -21013.985} C_VEL
LIN {X 0,Y 210.296,Z 429.464,A -85,B 0,C 180,E1 -21014.845,E2 -21014.845} C_VEL
LIN {X 0,Y 208.443,Z 426.691,A -85,B 0,C 180,E1 -21015.512,E2 -21015.512} C_VEL
LIN {X 0,Y 207.804,Z 424.497,A -85,B 0,C 180,E1 -21015.851,E2 -21015.851} C_VEL
LIN {X 0,Y 207.444,Z 422.001,A -85,B 0,C 180,E1 -21019.932,E2 -21019.932} C_VEL
LIN {X 0,Y 207.054,Z 419.309,A -85,B 0,C 180,E1 -21024.758,E2 -21024.758} C_VEL
LIN {X 0,Y 206.765,Z 417.59,A -85,B 0,C 180,E1 -21028.185,E2 -21028.185} C_VEL
LIN {X 0,Y 206.765,Z 417.357,A -85,B 0,C 180,E1 -21032.098,E2 -21032.098} C_VEL
LIN {X 0,Y 206.755,Z 417.356,A -85,B 0,C 180,E1 -21036.604,E2 -21036.604} C_VEL
LIN {X 0,Y 206.874,Z 417.336,A -85,B 0,C 180,E1 -21042.197,E2 -21042.197} C_VEL
LIN {X 0,Y 206.915,Z 417.333,A -85,B 0,C 180,E1 -21046.246,E2 -21046.246} C_VEL
LIN {X 0,Y 207.134,Z 417.307,A -85,B 0,C 180,E1 -21050.233,E2 -21050.233} C_VEL
LIN {X 0,Y 207.19,Z 417.296,A -85,B 0,C 180,E1 -21052.202,E2 -21052.202} C_VEL
LIN {X 0,Y 207.385,Z 417.276,A -85,B 0,C 180,E1 -21058.058,E2 -21058.058} C_VEL
LIN {X 0,Y 207.52,Z 417.26,A -85,B 0,C 180,E1 -21060,E2 -21060} C_VEL
LIN {X 0,Y 207.088,Z 417.314,A -85,B 0,C 180,E1 -21063.892,E2 -21063.892} C_VEL
LIN {X 0,Y 207.19,Z 417.303,A -85,B 0,C 180,E1 -21067.798,E2 -21067.798} C_VEL
LIN {X 0,Y 206.985,Z 417.328,A -85,B 0,C 180,E1 -21071.755,E2 -21071.755} C_VEL
LIN {X 0,Y 206.869,Z 417.343,A -85,B 0,C 180,E1 -21075.771,E2 -21075.771} C_VEL
LIN {X 0,Y 206.785,Z 417.352,A -85,B 0,C 180,E1 -21079.869,E2 -21079.869} C_VEL
LIN {X 0,Y 206.765,Z 417.355,A -85,B 0,C 180,E1 -21084.072,E2 -21084.072} C_VEL
LIN {X 0,Y 206.738,Z 417.358,A -85,B 0,C 180,E1 -21088.42,E2 -21088.42} C_VEL
LIN {X 0,Y 206.707,Z 417.363,A -85,B 0,C 180,E1 -21092.956,E2 -21092.956} C_VEL
LIN {X 0,Y 206.723,Z 417.361,A -85,B 0,C 180,E1 -21095.32,E2 -21095.32} C_VEL
LIN {X 0,Y 207.061,Z 419.734,A -85,B 0,C 180,E1 -21100.158,E2 -21100.158} C_VEL
LIN {X 0,Y 207.353,Z 421.924,A -85,B 0,C 180,E1 -21104.113,E2 -21104.113} C_VEL
LIN {X 0,Y 208.481,Z 424.911,A -85,B 0,C 180,E1 -21104.604,E2 -21104.604} C_VEL
LIN {X 0,Y 210.339,Z 427.423,A -85,B 0,C 180,E1 -21105.272,E2 -21105.272} C_VEL
LIN {X 0,Y 212.174,Z 431.015,A -85,B 0,C 180,E1 -21106.024,E2 -21106.024} C_VEL
LIN {X 0,Y 215.453,Z 437.55,A -85,B 0,C 180,E1 -21107.395,E2 -21107.395} C_VEL
LIN {X 0,Y 218.857,Z 445.658,A -85,B 0,C 180,E1 -21108.994,E2 -21108.994} C_VEL
LIN {X 0,Y 221.971,Z 455.646,A -85,B 0,C 180,E1 -21110.869,E2 -21110.869} C_VEL
LIN {X 0,Y 224.629,Z 467.654,A -85,B 0,C 180,E1 -21113.125,E2 -21113.125} C_VEL
LIN {X 0,Y 225.961,Z 477.699,A -85,B 0,C 180,E1 -21115.074,E2 -21115.074} C_VEL
LIN {X 0,Y 226.353,Z 488.368,A -85,B 0,C 180,E1 -21117.262,E2 -21117.262} C_VEL
LIN {X 0,Y 223.136,Z 498.871,A -85,B 0,C 180,E1 -21119.215,E2 -21119.215} C_VEL
LIN {X 0,Y 219.773,Z 508.281,A -85,B 0,C 180,E1 -21121.336,E2 -21121.336} C_VEL
LIN {X 0,Y 216.384,Z 517.735,A -85,B 0,C 180,E1 -21123.994,E2 -21123.994} C_VEL
LIN {X 0,Y 212.834,Z 526.752,A -85,B 0,C 180,E1 -21127.171,E2 -21127.171} C_VEL
LIN {X 0,Y 210.102,Z 534.012,A -85,B 0,C 180,E1 -21130.458,E2 -21130.458} C_VEL
LIN {X 0,Y 208.121,Z 539.096,A -85,B 0,C 180,E1 -21133.32,E2 -21133.32} C_VEL
LIN {X 0,Y 206.192,Z 544.362,A -85,B 0,C 180,E1 -21137.2,E2 -21137.2} C_VEL
LIN {X 0,Y 205.247,Z 547.301,A -85,B 0,C 180,E1 -21140.142,E2 -21140.142} C_VEL
LIN {X 0,Y 204.574,Z 549.997,A -85,B 0,C 180,E1 -21144.085,E2 -21144.085} C_VEL
LIN {X 0,Y 204.31,Z 551.344,A -85,B 0,C 180,E1 -21148.029,E2 -21148.029} C_VEL
LIN {X 0,Y 204.343,Z 551.521,A -85,B 0,C 180,E1 -21150,E2 -21150} C_VEL
LIN {X 0,Y 204.366,Z 550.888,A -85,B 0,C 180,E1 -21153.944,E2 -21153.944} C_VEL
LIN {X 0,Y 204.843,Z 548.918,A -85,B 0,C 180,E1 -21157.888,E2 -21157.888} C_VEL
LIN {X 0,Y 205.793,Z 545.568,A -85,B 0,C 180,E1 -21161.824,E2 -21161.824} C_VEL
LIN {X 0,Y 207.469,Z 540.735,A -85,B 0,C 180,E1 -21165.724,E2 -21165.724} C_VEL
LIN {X 0,Y 209.411,Z 536.067,A -85,B 0,C 180,E1 -21168.592,E2 -21168.592} C_VEL
LIN {X 0,Y 211.687,Z 529.939,A -85,B 0,C 180,E1 -21171.627,E2 -21171.627} C_VEL
LIN {X 0,Y 214.702,Z 522.205,A -85,B 0,C 180,E1 -21174.668,E2 -21174.668} C_VEL
LIN {X 0,Y 217.945,Z 513.68,A -85,B 0,C 180,E1 -21177.356,E2 -21177.356} C_VEL
LIN {X 0,Y 221.699,Z 503.343,A -85,B 0,C 180,E1 -21179.953,E2 -21179.953} C_VEL
LIN {X 0,Y 225.091,Z 492.952,A -85,B 0,C 180,E1 -21182.059,E2 -21182.059} C_VEL
LIN {X 0,Y 226.406,Z 488.468,A -85,B 0,C 180,E1 -21182.853,E2 -21182.853} C_VEL
LIN {X 0,Y 226.126,Z 479.975,A -85,B 0,C 180,E1 -21184.609,E2 -21184.609} C_VEL
LIN {X 0,Y 224.883,Z 468.882,A -85,B 0,C 180,E1 -21186.781,E2 -21186.781} C_VEL
LIN {X 0,Y 222.42,Z 457.054,A -85,B 0,C 180,E1 -21189.011,E2 -21189.011} C_VEL
LIN {X 0,Y 218.836,Z 445.553,A -85,B 0,C 180,E1 -21191.183,E2 -21191.183} C_VEL
LIN {X 0,Y 214.727,Z 435.755,A -85,B 0,C 180,E1 -21193.108,E2 -21193.108} C_VEL
LIN {X 0,Y 212.126,Z 430.934,A -85,B 0,C 180,E1 -21194.165,E2 -21194.165} C_VEL
LIN {X 0,Y 209.88,Z 426.733,A -85,B 0,C 180,E1 -21195.076,E2 -21195.076} C_VEL
LIN {X 0,Y 207.974,Z 423.921,A -85,B 0,C 180,E1 -21195.771,E2 -21195.771} C_VEL
LIN {X 0,Y 207.338,Z 421.87,A -85,B 0,C 180,E1 -21196.104,E2 -21196.104} C_VEL
LIN {X 0,Y 206.969,Z 419.063,A -85,B 0,C 180,E1 -21201.353,E2 -21201.353} C_VEL
LIN {X 0,Y 206.734,Z 417.449,A -85,B 0,C 180,E1 -21204.695,E2 -21204.695} C_VEL
LIN {X 0,Y 206.726,Z 417.361,A -85,B 0,C 180,E1 -21209.339,E2 -21209.339} C_VEL
LIN {X 0,Y 206.736,Z 417.359,A -85,B 0,C 180,E1 -21213.772,E2 -21213.772} C_VEL
LIN {X 0,Y 206.761,Z 417.356,A -85,B 0,C 180,E1 -21218.043,E2 -21218.043} C_VEL
LIN {X 0,Y 206.876,Z 417.34,A -85,B 0,C 180,E1 -21222.197,E2 -21222.197} C_VEL
LIN {X 0,Y 206.917,Z 417.335,A -85,B 0,C 180,E1 -21226.246,E2 -21226.246} C_VEL
LIN {X 0,Y 207.136,Z 417.309,A -85,B 0,C 180,E1 -21230.233,E2 -21230.233} C_VEL
LIN {X 0,Y 207.192,Z 417.303,A -85,B 0,C 180,E1 -21232.202,E2 -21232.202} C_VEL
LIN {X 0,Y 207.385,Z 417.276,A -85,B 0,C 180,E1 -21238.058,E2 -21238.058} C_VEL
LIN {X 0,Y 207.518,Z 417.261,A -85,B 0,C 180,E1 -21240,E2 -21240} C_VEL
LIN {X 0,Y 207.386,Z 417.279,A -85,B 0,C 180,E1 -21241.942,E2 -21241.942} C_VEL
LIN {X 0,Y 207.192,Z 417.3,A -85,B 0,C 180,E1 -21247.798,E2 -21247.798} C_VEL
LIN {X 0,Y 206.986,Z 417.328,A -85,B 0,C 180,E1 -21251.755,E2 -21251.755} C_VEL
LIN {X 0,Y 206.87,Z 417.342,A -85,B 0,C 180,E1 -21255.77,E2 -21255.77} C_VEL
LIN {X 0,Y 206.786,Z 417.353,A -85,B 0,C 180,E1 -21259.869,E2 -21259.869} C_VEL
LIN {X 0,Y 206.766,Z 417.346,A -85,B 0,C 180,E1 -21264.072,E2 -21264.072} C_VEL
LIN {X 0,Y 206.746,Z 417.356,A -85,B 0,C 180,E1 -21268.418,E2 -21268.418} C_VEL
LIN {X 0,Y 206.775,Z 417.648,A -85,B 0,C 180,E1 -21271.819,E2 -21271.819} C_VEL
LIN {X 0,Y 207.047,Z 419.479,A -85,B 0,C 180,E1 -21275.446,E2 -21275.446} C_VEL
LIN {X 0,Y 207.45,Z 422.061,A -85,B 0,C 180,E1 -21280.067,E2 -21280.067} C_VEL
LIN {X 0,Y 207.825,Z 424.52,A -85,B 0,C 180,E1 -21284.104,E2 -21284.104} C_VEL
LIN {X 0,Y 208.962,Z 427.68,A -85,B 0,C 180,E1 -21284.604,E2 -21284.604} C_VEL
LIN {X 0,Y 210.868,Z 430.443,A -85,B 0,C 180,E1 -21285.296,E2 -21285.296} C_VEL
LIN {X 0,Y 212.819,Z 434.144,A -85,B 0,C 180,E1 -21286.079,E2 -21286.079} C_VEL
LIN {X 0,Y 216.972,Z 443.284,A -85,B 0,C 180,E1 -21287.876,E2 -21287.876} C_VEL
LIN {X 0,Y 219.835,Z 451.561,A -85,B 0,C 180,E1 -21289.4,E2 -21289.4} C_VEL
LIN {X 0,Y 222.553,Z 462.037,A -85,B 0,C 180,E1 -21291.27,E2 -21291.27} C_VEL
LIN {X 0,Y 224.672,Z 474.346,A -85,B 0,C 180,E1 -21293.534,E2 -21293.534} C_VEL
LIN {X 0,Y 225.556,Z 486.48,A -85,B 0,C 180,E1 -21295.885,E2 -21295.885} C_VEL
LIN {X 0,Y 225.613,Z 493.018,A -85,B 0,C 180,E1 -21297.253,E2 -21297.253} C_VEL
LIN {X 0,Y 222.644,Z 502.98,A -85,B 0,C 180,E1 -21299.139,E2 -21299.139} C_VEL
LIN {X 0,Y 218.686,Z 514.034,A -85,B 0,C 180,E1 -21301.704,E2 -21301.704} C_VEL
LIN {X 0,Y 215.322,Z 523.158,A -85,B 0,C 180,E1 -21304.375,E2 -21304.375} C_VEL
LIN {X 0,Y 213.891,Z 526.864,A -85,B 0,C 180,E1 -21305.64,E2 -21305.64} C_VEL
LIN {X 0,Y 211.937,Z 530.267,A -85,B 0,C 180,E1 -21306.843,E2 -21306.843} C_VEL
LIN {X 0,Y 207.231,Z 535.37,A -85,B 0,C 180,E1 -21308.781,E2 -21308.781} C_VEL
LIN {X 0,Y 202.734,Z 539.976,A -85,B 0,C 180,E1 -21310.89,E2 -21310.89} C_VEL
LIN {X 0,Y 201.148,Z 542.442,A -85,B 0,C 180,E1 -21312.333,E2 -21312.333} C_VEL
LIN {X 0,Y 199.28,Z 547.11,A -85,B 0,C 180,E1 -21315.707,E2 -21315.707} C_VEL
LIN {X 0,Y 197.983,Z 551.232,A -85,B 0,C 180,E1 -21319.776,E2 -21319.776} C_VEL
LIN {X 0,Y 197.337,Z 553.924,A -85,B 0,C 180,E1 -21323.866,E2 -21323.866} C_VEL
LIN {X 0,Y 197.187,Z 555.255,A -85,B 0,C 180,E1 -21327.957,E2 -21327.957} C_VEL
LIN {X 0,Y 197.244,Z 555.418,A -85,B 0,C 180,E1 -21330,E2 -21330} C_VEL
LIN {X 0,Y 197.176,Z 554.74,A -85,B 0,C 180,E1 -21334.088,E2 -21334.088} C_VEL
LIN {X 0,Y 197.582,Z 552.719,A -85,B 0,C 180,E1 -21338.18,E2 -21338.18} C_VEL
LIN {X 0,Y 198.555,Z 549.306,A -85,B 0,C 180,E1 -21342.261,E2 -21342.261} C_VEL
LIN {X 0,Y 200.341,Z 544.401,A -85,B 0,C 180,E1 -21346.298,E2 -21346.298} C_VEL
LIN {X 0,Y 202.979,Z 537.859,A -85,B 0,C 180,E1 -21350.258,E2 -21350.258} C_VEL
LIN {X 0,Y 205.804,Z 530.578,A -85,B 0,C 180,E1 -21353.656,E2 -21353.656} C_VEL
LIN {X 0,Y 209.478,Z 521.56,A -85,B 0,C 180,E1 -21356.931,E2 -21356.931} C_VEL
LIN {X 0,Y 213.096,Z 512.099,A -85,B 0,C 180,E1 -21359.65,E2 -21359.65} C_VEL
LIN {X 0,Y 216.918,Z 501.625,A -85,B 0,C 180,E1 -21362.042,E2 -21362.042} C_VEL
LIN {X 0,Y 219.236,Z 493.906,A -85,B 0,C 180,E1 -21363.543,E2 -21363.543} C_VEL
LIN {X 0,Y 219.032,Z 483.693,A -85,B 0,C 180,E1 -21365.755,E2 -21365.755} C_VEL
LIN {X 0,Y 218.101,Z 473.244,A -85,B 0,C 180,E1 -21367.858,E2 -21367.858} C_VEL
LIN {X 0,Y 216.018,Z 461.434,A -85,B 0,C 180,E1 -21370.134,E2 -21370.134} C_VEL
LIN {X 0,Y 212.842,Z 449.745,A -85,B 0,C 180,E1 -21372.369,E2 -21372.369} C_VEL
LIN {X 0,Y 209.337,Z 441.247,A -85,B 0,C 180,E1 -21374.146,E2 -21374.146} C_VEL
LIN {X 0,Y 205.943,Z 434.318,A -85,B 0,C 180,E1 -21375.687,E2 -21375.687} C_VEL
LIN {X 0,Y 203.928,Z 430.696,A -85,B 0,C 180,E1 -21376.551,E2 -21376.551} C_VEL
LIN {X 0,Y 203.316,Z 429.485,A -85,B 0,C 180,E1 -21376.826,E2 -21376.826} C_VEL
LIN {X 0,Y 201.283,Z 426.525,A -85,B 0,C 180,E1 -21377.63,E2 -21377.63} C_VEL
LIN {X 0,Y 200.647,Z 424.407,A -85,B 0,C 180,E1 -21377.997,E2 -21377.997} C_VEL
LIN {X 0,Y 200.374,Z 422.767,A -85,B 0,C 180,E1 -21380.851,E2 -21380.851} C_VEL
LIN {X 0,Y 199.961,Z 420.186,A -85,B 0,C 180,E1 -21385.782,E2 -21385.782} C_VEL
LIN {X 0,Y 199.812,Z 419.038,A -85,B 0,C 180,E1 -21388.157,E2 -21388.157} C_VEL
LIN {X 0,Y 199.665,Z 418.241,A -85,B 0,C 180,E1 -21390.476,E2 -21390.476} C_VEL
LIN {X 0,Y 199.665,Z 418.24,A -85,B 0,C 180,E1 -21395.015,E2 -21395.015} C_VEL
LIN {X 0,Y 199.692,Z 418.236,A -85,B 0,C 180,E1 -21399.394,E2 -21399.394} C_VEL
LIN {X 0,Y 199.806,Z 418.222,A -85,B 0,C 180,E1 -21403.657,E2 -21403.657} C_VEL
LIN {X 0,Y 200.069,Z 418.183,A -85,B 0,C 180,E1 -21409.603,E2 -21409.603} C_VEL
LIN {X 0,Y 200.134,Z 418.176,A -85,B 0,C 180,E1 -21411.925,E2 -21411.925} C_VEL
LIN {X 0,Y 200.324,Z 418.156,A -85,B 0,C 180,E1 -21417.99,E2 -21417.99} C_VEL
LIN {X 0,Y 200.484,Z 418.136,A -85,B 0,C 180,E1 -21420,E2 -21420} C_VEL
LIN {X 0,Y 200.034,Z 418.192,A -85,B 0,C 180,E1 -21424.03,E2 -21424.03} C_VEL
LIN {X 0,Y 200.134,Z 418.181,A -85,B 0,C 180,E1 -21428.075,E2 -21428.075} C_VEL
LIN {X 0,Y 199.916,Z 418.208,A -85,B 0,C 180,E1 -21432.177,E2 -21432.177} C_VEL
LIN {X 0,Y 199.807,Z 418.218,A -85,B 0,C 180,E1 -21436.344,E2 -21436.344} C_VEL
LIN {X 0,Y 199.702,Z 418.235,A -85,B 0,C 180,E1 -21440.605,E2 -21440.605} C_VEL
LIN {X 0,Y 199.674,Z 418.238,A -85,B 0,C 180,E1 -21444.984,E2 -21444.984} C_VEL
LIN {X 0,Y 199.666,Z 418.239,A -85,B 0,C 180,E1 -21449.524,E2 -21449.524} C_VEL
LIN {X 0,Y 199.659,Z 418.24,A -85,B 0,C 180,E1 -21452.35,E2 -21452.35} C_VEL
LIN {X 0,Y 199.657,Z 418.304,A -85,B 0,C 180,E1 -21454.278,E2 -21454.278} C_VEL
LIN {X 0,Y 200.023,Z 420.672,A -85,B 0,C 180,E1 -21459.377,E2 -21459.377} C_VEL
LIN {X 0,Y 200.196,Z 422.024,A -85,B 0,C 180,E1 -21461.956,E2 -21461.956} C_VEL
LIN {X 0,Y 201.345,Z 425.02,A -85,B 0,C 180,E1 -21462.504,E2 -21462.504} C_VEL
LIN {X 0,Y 203.46,Z 427.878,A -85,B 0,C 180,E1 -21463.346,E2 -21463.346} C_VEL
LIN {X 0,Y 205.535,Z 431.605,A -85,B 0,C 180,E1 -21464.247,E2 -21464.247} C_VEL
LIN {X 0,Y 210.104,Z 440.445,A -85,B 0,C 180,E1 -21466.304,E2 -21466.304} C_VEL
LIN {X 0,Y 213.899,Z 450.296,A -85,B 0,C 180,E1 -21468.374,E2 -21468.374} C_VEL
LIN {X 0,Y 216.74,Z 460.244,A -85,B 0,C 180,E1 -21470.364,E2 -21470.364} C_VEL
LIN {X 0,Y 218.911,Z 471.607,A -85,B 0,C 180,E1 -21472.639,E2 -21472.639} C_VEL
LIN {X 0,Y 219.88,Z 481.245,A -85,B 0,C 180,E1 -21474.649,E2 -21474.649} C_VEL
LIN {X 0,Y 220.147,Z 488.732,A -85,B 0,C 180,E1 -21476.281,E2 -21476.281} C_VEL
LIN {X 0,Y 217.42,Z 497.876,A -85,B 0,C 180,E1 -21478.041,E2 -21478.041} C_VEL
LIN {X 0,Y 213.547,Z 508.353,A -85,B 0,C 180,E1 -21480.419,E2 -21480.419} C_VEL
LIN {X 0,Y 210.01,Z 517.807,A -85,B 0,C 180,E1 -21483.142,E2 -21483.142} C_VEL
LIN {X 0,Y 206.28,Z 526.822,A -85,B 0,C 180,E1 -21486.402,E2 -21486.402} C_VEL
LIN {X 0,Y 204.117,Z 532.206,A -85,B 0,C 180,E1 -21488.833,E2 -21488.833} C_VEL
LIN {X 0,Y 201.998,Z 537.559,A -85,B 0,C 180,E1 -21491.752,E2 -21491.752} C_VEL
LIN {X 0,Y 199.646,Z 543.243,A -85,B 0,C 180,E1 -21495.735,E2 -21495.735} C_VEL
LIN {X 0,Y 198.229,Z 547.37,A -85,B 0,C 180,E1 -21499.789,E2 -21499.789} C_VEL
LIN {X 0,Y 197.507,Z 550.066,A -85,B 0,C 180,E1 -21503.872,E2 -21503.872} C_VEL
LIN {X 0,Y 197.221,Z 551.413,A -85,B 0,C 180,E1 -21507.958,E2 -21507.958} C_VEL
LIN {X 0,Y 197.25,Z 551.59,A -85,B 0,C 180,E1 -21510,E2 -21510} C_VEL
LIN {X 0,Y 197.286,Z 550.956,A -85,B 0,C 180,E1 -21514.086,E2 -21514.086} C_VEL
LIN {X 0,Y 197.78,Z 548.987,A -85,B 0,C 180,E1 -21518.172,E2 -21518.172} C_VEL
LIN {X 0,Y 198.824,Z 545.636,A -85,B 0,C 180,E1 -21522.245,E2 -21522.245} C_VEL
LIN {X 0,Y 200.628,Z 540.803,A -85,B 0,C 180,E1 -21526.275,E2 -21526.275} C_VEL
LIN {X 0,Y 202.662,Z 536.135,A -85,B 0,C 180,E1 -21529.235,E2 -21529.235} C_VEL
LIN {X 0,Y 205.329,Z 529.351,A -85,B 0,C 180,E1 -21532.648,E2 -21532.648} C_VEL
LIN {X 0,Y 208.259,Z 522.272,A -85,B 0,C 180,E1 -21535.485,E2 -21535.485} C_VEL
LIN {X 0,Y 211.658,Z 513.746,A -85,B 0,C 180,E1 -21538.24,E2 -21538.24} C_VEL
LIN {X 0,Y 215.555,Z 503.408,A -85,B 0,C 180,E1 -21540.899,E2 -21540.899} C_VEL
LIN {X 0,Y 219.105,Z 493.017,A -85,B 0,C 180,E1 -21543.045,E2 -21543.045} C_VEL
LIN {X 0,Y 220.023,Z 489.98,A -85,B 0,C 180,E1 -21543.598,E2 -21543.598} C_VEL
LIN {X 0,Y 220.014,Z 483.146,A -85,B 0,C 180,E1 -21545.099,E2 -21545.099} C_VEL
LIN {X 0,Y 219.052,Z 472.319,A -85,B 0,C 180,E1 -21547.356,E2 -21547.356} C_VEL
LIN {X 0,Y 216.92,Z 460.661,A -85,B 0,C 180,E1 -21549.693,E2 -21549.693} C_VEL
LIN {X 0,Y 213.709,Z 449.601,A -85,B 0,C 180,E1 -21551.923,E2 -21551.923} C_VEL
LIN {X 0,Y 209.635,Z 439.475,A -85,B 0,C 180,E1 -21554.089,E2 -21554.089} C_VEL
LIN {X 0,Y 205.497,Z 431.545,A -85,B 0,C 180,E1 -21555.947,E2 -21555.947} C_VEL
LIN {X 0,Y 203.516,Z 428.004,A -85,B 0,C 180,E1 -21556.808,E2 -21556.808} C_VEL
LIN {X 0,Y 202.699,Z 426.777,A -85,B 0,C 180,E1 -21557.151,E2 -21557.151} C_VEL
LIN {X 0,Y 200.738,Z 423.851,A -85,B 0,C 180,E1 -21557.944,E2 -21557.944} C_VEL
LIN {X 0,Y 200.173,Z 421.982,A -85,B 0,C 180,E1 -21558.242,E2 -21558.242} C_VEL
LIN {X 0,Y 200.042,Z 420.693,A -85,B 0,C 180,E1 -21560.773,E2 -21560.773} C_VEL
LIN {X 0,Y 199.657,Z 418.404,A -85,B 0,C 180,E1 -21565.722,E2 -21565.722} C_VEL
LIN {X 0,Y 199.703,Z 418.232,A -85,B 0,C 180,E1 -21568.137,E2 -21568.137} C_VEL
LIN {X 0,Y 199.69,Z 418.236,A -85,B 0,C 180,E1 -21572.772,E2 -21572.772} C_VEL
LIN {X 0,Y 199.741,Z 418.228,A -85,B 0,C 180,E1 -21577.229,E2 -21577.229} C_VEL
LIN {X 0,Y 199.799,Z 418.223,A -85,B 0,C 180,E1 -21581.757,E2 -21581.757} C_VEL
LIN {X 0,Y 199.851,Z 418.216,A -85,B 0,C 180,E1 -21585.749,E2 -21585.749} C_VEL
LIN {X 0,Y 200.078,Z 418.188,A -85,B 0,C 180,E1 -21589.884,E2 -21589.884} C_VEL
LIN {X 0,Y 200.135,Z 418.18,A -85,B 0,C 180,E1 -21591.925,E2 -21591.925} C_VEL
LIN {X 0,Y 200.325,Z 418.156,A -85,B 0,C 180,E1 -21597.989,E2 -21597.989} C_VEL
LIN {X 0,Y 200.482,Z 418.138,A -85,B 0,C 180,E1 -21600,E2 -21600} C_VEL
LIN {X 0,Y 200.036,Z 418.193,A -85,B 0,C 180,E1 -21604.029,E2 -21604.029} C_VEL
LIN {X 0,Y 200.135,Z 418.179,A -85,B 0,C 180,E1 -21608.075,E2 -21608.075} C_VEL
LIN {X 0,Y 199.917,Z 418.207,A -85,B 0,C 180,E1 -21612.177,E2 -21612.177} C_VEL
LIN {X 0,Y 199.807,Z 418.221,A -85,B 0,C 180,E1 -21616.343,E2 -21616.343} C_VEL
LIN {X 0,Y 199.703,Z 418.234,A -85,B 0,C 180,E1 -21620.605,E2 -21620.605} C_VEL
LIN {X 0,Y 199.675,Z 418.233,A -85,B 0,C 180,E1 -21624.984,E2 -21624.984} C_VEL
LIN {X 0,Y 199.677,Z 418.234,A -85,B 0,C 180,E1 -21629.522,E2 -21629.522} C_VEL
LIN {X 0,Y 199.844,Z 419.376,A -85,B 0,C 180,E1 -21632.433,E2 -21632.433} C_VEL
LIN {X 0,Y 200.167,Z 421.477,A -85,B 0,C 180,E1 -21636.647,E2 -21636.647} C_VEL
LIN {X 0,Y 200.68,Z 424.401,A -85,B 0,C 180,E1 -21641.903,E2 -21641.903} C_VEL
LIN {X 0,Y 201.971,Z 427.792,A -85,B 0,C 180,E1 -21642.567,E2 -21642.567} C_VEL
LIN {X 0,Y 203.824,Z 430.276,A -85,B 0,C 180,E1 -21643.295,E2 -21643.295} C_VEL
LIN {X 0,Y 205.731,Z 434.029,A -85,B 0,C 180,E1 -21644.143,E2 -21644.143} C_VEL
LIN {X 0,Y 206.819,Z 435.967,A -85,B 0,C 180,E1 -21644.6,E2 -21644.6} C_VEL
LIN {X 0,Y 210.349,Z 443.206,A -85,B 0,C 180,E1 -21646.222,E2 -21646.222} C_VEL
LIN {X 0,Y 214.069,Z 453.631,A -85,B 0,C 180,E1 -21648.322,E2 -21648.322} C_VEL
LIN {X 0,Y 216.708,Z 464.349,A -85,B 0,C 180,E1 -21650.374,E2 -21650.374} C_VEL
LIN {X 0,Y 218.478,Z 475.171,A -85,B 0,C 180,E1 -21652.479,E2 -21652.479} C_VEL
LIN {X 0,Y 219.237,Z 486.41,A -85,B 0,C 180,E1 -21654.759,E2 -21654.759} C_VEL
LIN {X 0,Y 219.259,Z 494.102,A -85,B 0,C 180,E1 -21656.448,E2 -21656.448} C_VEL
LIN {X 0,Y 216.573,Z 502.915,A -85,B 0,C 180,E1 -21658.175,E2 -21658.175} C_VEL
LIN {X 0,Y 212.445,Z 513.967,A -85,B 0,C 180,E1 -21660.794,E2 -21660.794} C_VEL
LIN {X 0,Y 208.924,Z 523.091,A -85,B 0,C 180,E1 -21663.53,E2 -21663.53} C_VEL
LIN {X 0,Y 205.347,Z 531.811,A -85,B 0,C 180,E1 -21666.822,E2 -21666.822} C_VEL
LIN {X 0,Y 202.895,Z 537.951,A -85,B 0,C 180,E1 -21669.733,E2 -21669.733} C_VEL
LIN {X 0,Y 201.148,Z 542.442,A -85,B 0,C 180,E1 -21672.333,E2 -21672.333} C_VEL
LIN {X 0,Y 199.639,Z 544.762,A -85,B 0,C 180,E1 -21673.825,E2 -21673.825} C_VEL
LIN {X 0,Y 195.589,Z 548.034,A -85,B 0,C 180,E1 -21676.273,E2 -21676.273} C_VEL
LIN {X 0,Y 192.401,Z 550.216,A -85,B 0,C 180,E1 -21678.335,E2 -21678.335} C_VEL
LIN {X 0,Y 190.902,Z 551.638,A -85,B 0,C 180,E1 -21680,E2 -21680} C_VEL
LIN {X 0,Y 190.691,Z 552.01,A -85,B 0,C 180,E1 -21680.576,E2 -21680.576} C_VEL
LIN {X 0,Y 190.275,Z 553.856,A -85,B 0,C 180,E1 -21683.638,E2 -21683.638} C_VEL
LIN {X 0,Y 190.083,Z 555.186,A -85,B 0,C 180,E1 -21687.881,E2 -21687.881} C_VEL
LIN {X 0,Y 190.152,Z 555.349,A -85,B 0,C 180,E1 -21690,E2 -21690} C_VEL
LIN {X 0,Y 190.089,Z 554.671,A -85,B 0,C 180,E1 -21694.24,E2 -21694.24} C_VEL
LIN {X 0,Y 190.529,Z 552.649,A -85,B 0,C 180,E1 -21698.485,E2 -21698.485} C_VEL
LIN {X 0,Y 191.592,Z 549.236,A -85,B 0,C 180,E1 -21702.714,E2 -21702.714} C_VEL
LIN {X 0,Y 193.497,Z 544.33,A -85,B 0,C 180,E1 -21706.892,E2 -21706.892} C_VEL
LIN {X 0,Y 196.278,Z 537.788,A -85,B 0,C 180,E1 -21710.981,E2 -21710.981} C_VEL
LIN {X 0,Y 199.275,Z 530.507,A -85,B 0,C 180,E1 -21714.481,E2 -21714.481} C_VEL
LIN {X 0,Y 203.14,Z 521.488,A -85,B 0,C 180,E1 -21717.843,E2 -21717.843} C_VEL
LIN {X 0,Y 206.951,Z 512.027,A -85,B 0,C 180,E1 -21720.623,E2 -21720.623} C_VEL
LIN {X 0,Y 210.911,Z 501.587,A -85,B 0,C 180,E1 -21723.06,E2 -21723.06} C_VEL
LIN {X 0,Y 212.89,Z 495.069,A -85,B 0,C 180,E1 -21724.38,E2 -21724.38} C_VEL
LIN {X 0,Y 212.856,Z 484.993,A -85,B 0,C 180,E1 -21726.677,E2 -21726.677} C_VEL
LIN {X 0,Y 211.933,Z 473.802,A -85,B 0,C 180,E1 -21729.055,E2 -21729.055} C_VEL
LIN {X 0,Y 209.874,Z 461.98,A -85,B 0,C 180,E1 -21731.473,E2 -21731.473} C_VEL
LIN {X 0,Y 207.259,Z 452.406,A -85,B 0,C 180,E1 -21733.441,E2 -21733.441} C_VEL
LIN {X 0,Y 203.503,Z 443.017,A -85,B 0,C 180,E1 -21735.578,E2 -21735.578} C_VEL
LIN {X 0,Y 200.813,Z 437.836,A -85,B 0,C 180,E1 -21736.883,E2 -21736.883} C_VEL
LIN {X 0,Y 198.95,Z 434.271,A -85,B 0,C 180,E1 -21737.784,E2 -21737.784} C_VEL
LIN {X 0,Y 196.936,Z 430.575,A -85,B 0,C 180,E1 -21738.744,E2 -21738.744} C_VEL
LIN {X 0,Y 196.175,Z 429.425,A -85,B 0,C 180,E1 -21739.093,E2 -21739.093} C_VEL
LIN {X 0,Y 194.251,Z 426.766,A -85,B 0,C 180,E1 -21739.931,E2 -21739.931} C_VEL
LIN {X 0,Y 193.454,Z 424.306,A -85,B 0,C 180,E1 -21740.411,E2 -21740.411} C_VEL
LIN {X 0,Y 193.111,Z 422.257,A -85,B 0,C 180,E1 -21744.388,E2 -21744.388} C_VEL
LIN {X 0,Y 192.736,Z 419.969,A -85,B 0,C 180,E1 -21749.303,E2 -21749.303} C_VEL
LIN {X 0,Y 192.661,Z 419.113,A -85,B 0,C 180,E1 -21751.691,E2 -21751.691} C_VEL
LIN {X 0,Y 192.686,Z 419.109,A -85,B 0,C 180,E1 -21756.346,E2 -21756.346} C_VEL
LIN {X 0,Y 192.732,Z 419.1,A -85,B 0,C 180,E1 -21761.458,E2 -21761.458} C_VEL
LIN {X 0,Y 192.773,Z 419.092,A -85,B 0,C 180,E1 -21765.215,E2 -21765.215} C_VEL
LIN {X 0,Y 193.021,Z 419.061,A -85,B 0,C 180,E1 -21769.511,E2 -21769.511} C_VEL
LIN {X 0,Y 193.007,Z 419.063,A -85,B 0,C 180,E1 -21773.729,E2 -21773.729} C_VEL
LIN {X 0,Y 193.266,Z 419.035,A -85,B 0,C 180,E1 -21777.916,E2 -21777.916} C_VEL
LIN {X 0,Y 193.448,Z 419.012,A -85,B 0,C 180,E1 -21780,E2 -21780} C_VEL
LIN {X 0,Y 192.981,Z 419.07,A -85,B 0,C 180,E1 -21784.177,E2 -21784.177} C_VEL
LIN {X 0,Y 193.081,Z 419.058,A -85,B 0,C 180,E1 -21788.372,E2 -21788.372} C_VEL
LIN {X 0,Y 192.855,Z 419.083,A -85,B 0,C 180,E1 -21792.63,E2 -21792.63} C_VEL
LIN {X 0,Y 192.76,Z 419.093,A -85,B 0,C 180,E1 -21796.959,E2 -21796.959} C_VEL
LIN {X 0,Y 192.638,Z 419.114,A -85,B 0,C 180,E1 -21801.397,E2 -21801.397} C_VEL
LIN {X 0,Y 192.665,Z 419.111,A -85,B 0,C 180,E1 -21804.225,E2 -21804.225} C_VEL
LIN {X 0,Y 192.645,Z 419.113,A -85,B 0,C 180,E1 -21808.889,E2 -21808.889} C_VEL
LIN {X 0,Y 192.605,Z 419.276,A -85,B 0,C 180,E1 -21813.185,E2 -21813.185} C_VEL
LIN {X 0,Y 192.852,Z 420.771,A -85,B 0,C 180,E1 -21816.704,E2 -21816.704} C_VEL
LIN {X 0,Y 193.077,Z 422.172,A -85,B 0,C 180,E1 -21819.549,E2 -21819.549} C_VEL
LIN {X 0,Y 194.196,Z 425.112,A -85,B 0,C 180,E1 -21820.147,E2 -21820.147} C_VEL
LIN {X 0,Y 196.412,Z 427.86,A -85,B 0,C 180,E1 -21821.11,E2 -21821.11} C_VEL
LIN {X 0,Y 198.387,Z 431.602,A -85,B 0,C 180,E1 -21822.075,E2 -21822.075} C_VEL
LIN {X 0,Y 199.593,Z 433.451,A -85,B 0,C 180,E1 -21822.613,E2 -21822.613} C_VEL
LIN {X 0,Y 204.048,Z 442.042,A -85,B 0,C 180,E1 -21824.83,E2 -21824.83} C_VEL
LIN {X 0,Y 207.585,Z 450.759,A -85,B 0,C 180,E1 -21826.853,E2 -21826.853} C_VEL
LIN {X 0,Y 210.652,Z 461.421,A -85,B 0,C 180,E1 -21829.153,E2 -21829.153} C_VEL
LIN {X 0,Y 212.628,Z 471.718,A -85,B 0,C 180,E1 -21831.34,E2 -21831.34} C_VEL
LIN {X 0,Y 213.693,Z 482.48,A -85,B 0,C 180,E1 -21833.702,E2 -21833.702} C_VEL
LIN {X 0,Y 213.739,Z 490.833,A -85,B 0,C 180,E1 -21835.621,E2 -21835.621} C_VEL
LIN {X 0,Y 210.273,Z 501.004,A -85,B 0,C 180,E1 -21837.672,E2 -21837.672} C_VEL
LIN {X 0,Y 206.737,Z 510.131,A -85,B 0,C 180,E1 -21839.906,E2 -21839.906} C_VEL
LIN {X 0,Y 203.082,Z 519.274,A -85,B 0,C 180,E1 -21842.707,E2 -21842.707} C_VEL
LIN {X 0,Y 199.769,Z 526.893,A -85,B 0,C 180,E1 -21845.583,E2 -21845.583} C_VEL
LIN {X 0,Y 196.683,Z 534.154,A -85,B 0,C 180,E1 -21849.064,E2 -21849.064} C_VEL
LIN {X 0,Y 194.541,Z 539.237,A -85,B 0,C 180,E1 -21852.117,E2 -21852.117} C_VEL
LIN {X 0,Y 192.727,Z 543.314,A -85,B 0,C 180,E1 -21855.211,E2 -21855.211} C_VEL
LIN {X 0,Y 191.233,Z 547.44,A -85,B 0,C 180,E1 -21859.412,E2 -21859.412} C_VEL
LIN {X 0,Y 190.426,Z 550.136,A -85,B 0,C 180,E1 -21863.643,E2 -21863.643} C_VEL
LIN {X 0,Y 190.135,Z 551.482,A -85,B 0,C 180,E1 -21867.882,E2 -21867.882} C_VEL
LIN {X 0,Y 190.159,Z 551.659,A -85,B 0,C 180,E1 -21870,E2 -21870} C_VEL
LIN {X 0,Y 190.2,Z 551.025,A -85,B 0,C 180,E1 -21874.238,E2 -21874.238} C_VEL
LIN {X 0,Y 190.736,Z 549.055,A -85,B 0,C 180,E1 -21878.476,E2 -21878.476} C_VEL
LIN {X 0,Y 191.851,Z 545.704,A -85,B 0,C 180,E1 -21882.697,E2 -21882.697} C_VEL
LIN {X 0,Y 193.812,Z 540.87,A -85,B 0,C 180,E1 -21886.864,E2 -21886.864} C_VEL
LIN {X 0,Y 195.925,Z 536.203,A -85,B 0,C 180,E1 -21889.924,E2 -21889.924} C_VEL
LIN {X 0,Y 198.769,Z 529.419,A -85,B 0,C 180,E1 -21893.439,E2 -21893.439} C_VEL
LIN {X 0,Y 201.847,Z 522.339,A -85,B 0,C 180,E1 -21896.356,E2 -21896.356} C_VEL
LIN {X 0,Y 205.43,Z 513.812,A -85,B 0,C 180,E1 -21899.177,E2 -21899.177} C_VEL
LIN {X 0,Y 209.483,Z 503.474,A -85,B 0,C 180,E1 -21901.898,E2 -21901.898} C_VEL
LIN {X 0,Y 213.159,Z 493.083,A -85,B 0,C 180,E1 -21904.091,E2 -21904.091} C_VEL
LIN {X 0,Y 213.774,Z 491.145,A -85,B 0,C 180,E1 -21904.45,E2 -21904.45} C_VEL
LIN {X 0,Y 213.709,Z 483.216,A -85,B 0,C 180,E1 -21906.296,E2 -21906.296} C_VEL
LIN {X 0,Y 212.936,Z 473.642,A -85,B 0,C 180,E1 -21908.383,E2 -21908.383} C_VEL
LIN {X 0,Y 211.012,Z 462.616,A -85,B 0,C 180,E1 -21910.737,E2 -21910.737} C_VEL
LIN {X 0,Y 208.025,Z 451.859,A -85,B 0,C 180,E1 -21913.064,E2 -21913.064} C_VEL
LIN {X 0,Y 204.439,Z 442.941,A -85,B 0,C 180,E1 -21915.134,E2 -21915.134} C_VEL
LIN {X 0,Y 200.88,Z 435.899,A -85,B 0,C 180,E1 -21916.929,E2 -21916.929} C_VEL
LIN {X 0,Y 198.706,Z 432.002,A -85,B 0,C 180,E1 -21917.978,E2 -21917.978} C_VEL
LIN {X 0,Y 196.654,Z 428.53,A -85,B 0,C 180,E1 -21918.944,E2 -21918.944} C_VEL
LIN {X 0,Y 196.041,Z 427.318,A -85,B 0,C 180,E1 -21919.255,E2 -21919.255} C_VEL
LIN {X 0,Y 193.969,Z 424.653,A -85,B 0,C 180,E1 -21920.162,E2 -21920.162} C_VEL
LIN {X 0,Y 193.063,Z 422.063,A -85,B 0,C 180,E1 -21920.706,E2 -21920.706} C_VEL
LIN {X 0,Y 192.787,Z 420.419,A -85,B 0,C 180,E1 -21924.318,E2 -21924.318} C_VEL
LIN {X 0,Y 192.61,Z 419.272,A -85,B 0,C 180,E1 -21927.059,E2 -21927.059} C_VEL
LIN {X 0,Y 192.667,Z 419.112,A -85,B 0,C 180,E1 -21931.692,E2 -21931.692} C_VEL
LIN {X 0,Y 192.709,Z 419.1,A -85,B 0,C 180,E1 -21936.349,E2 -21936.349} C_VEL
LIN {X 0,Y 192.735,Z 419.103,A -85,B 0,C 180,E1 -21941.457,E2 -21941.457} C_VEL
LIN {X 0,Y 192.775,Z 419.097,A -85,B 0,C 180,E1 -21945.214,E2 -21945.214} C_VEL
LIN {X 0,Y 193.023,Z 419.067,A -85,B 0,C 180,E1 -21949.511,E2 -21949.511} C_VEL
LIN {X 0,Y 193.008,Z 419.067,A -85,B 0,C 180,E1 -21953.728,E2 -21953.728} C_VEL
LIN {X 0,Y 193.267,Z 419.035,A -85,B 0,C 180,E1 -21957.916,E2 -21957.916} C_VEL
LIN {X 0,Y 193.446,Z 419.014,A -85,B 0,C 180,E1 -21960,E2 -21960} C_VEL
LIN {X 0,Y 192.983,Z 419.072,A -85,B 0,C 180,E1 -21964.177,E2 -21964.177} C_VEL
LIN {X 0,Y 193.082,Z 419.058,A -85,B 0,C 180,E1 -21968.372,E2 -21968.372} C_VEL
LIN {X 0,Y 192.856,Z 419.086,A -85,B 0,C 180,E1 -21972.63,E2 -21972.63} C_VEL
LIN {X 0,Y 192.76,Z 419.097,A -85,B 0,C 180,E1 -21976.958,E2 -21976.958} C_VEL
LIN {X 0,Y 192.639,Z 419.113,A -85,B 0,C 180,E1 -21981.397,E2 -21981.397} C_VEL
LIN {X 0,Y 192.666,Z 419.102,A -85,B 0,C 180,E1 -21984.225,E2 -21984.225} C_VEL
LIN {X 0,Y 192.688,Z 419.253,A -85,B 0,C 180,E1 -21988.911,E2 -21988.911} C_VEL
LIN {X 0,Y 192.923,Z 421.117,A -85,B 0,C 180,E1 -21993.123,E2 -21993.123} C_VEL
LIN {X 0,Y 193.222,Z 422.934,A -85,B 0,C 180,E1 -21996.85,E2 -21996.85} C_VEL
LIN {X 0,Y 193.473,Z 424.411,A -85,B 0,C 180,E1 -21999.528,E2 -21999.528} C_VEL
LIN {X 0,Y 194.534,Z 427.28,A -85,B 0,C 180,E1 -22000.096,E2 -22000.096} C_VEL
LIN {X 0,Y 196.925,Z 430.427,A -85,B 0,C 180,E1 -22001.139,E2 -22001.139} C_VEL
LIN {X 0,Y 198.813,Z 434.042,A -85,B 0,C 180,E1 -22002.056,E2 -22002.056} C_VEL
LIN {X 0,Y 199.999,Z 436.04,A -85,B 0,C 180,E1 -22002.596,E2 -22002.596} C_VEL
LIN {X 0,Y 204.367,Z 444.832,A -85,B 0,C 180,E1 -22004.787,E2 -22004.787} C_VEL
LIN {X 0,Y 208.007,Z 454.531,A -85,B 0,C 180,E1 -22006.941,E2 -22006.941} C_VEL
LIN {X 0,Y 210.857,Z 466.411,A -85,B 0,C 180,E1 -22009.381,E2 -22009.381} C_VEL
LIN {X 0,Y 212.463,Z 477.606,A -85,B 0,C 180,E1 -22011.7,E2 -22011.7} C_VEL
LIN {X 0,Y 213.03,Z 488.958,A -85,B 0,C 180,E1 -22014.156,E2 -22014.156} C_VEL
LIN {X 0,Y 212.726,Z 496.318,A -85,B 0,C 180,E1 -22015.83,E2 -22015.83} C_VEL
LIN {X 0,Y 209.073,Z 506.765,A -85,B 0,C 180,E1 -22018.032,E2 -22018.032} C_VEL
LIN {X 0,Y 204.96,Z 517.159,A -85,B 0,C 180,E1 -22020.749,E2 -22020.749} C_VEL
LIN {X 0,Y 201.424,Z 525.736,A -85,B 0,C 180,E1 -22023.585,E2 -22023.585} C_VEL
LIN {X 0,Y 197.875,Z 533.944,A -85,B 0,C 180,E1 -22027.002,E2 -22027.002} C_VEL
LIN {X 0,Y 195.46,Z 539.697,A -85,B 0,C 180,E1 -22030.026,E2 -22030.026} C_VEL
LIN {X 0,Y 193.498,Z 544.407,A -85,B 0,C 180,E1 -22033.108,E2 -22033.108} C_VEL
LIN {X 0,Y 191.6,Z 549.289,A -85,B 0,C 180,E1 -22037.286,E2 -22037.286} C_VEL
LIN {X 0,Y 190.691,Z 552.01,A -85,B 0,C 180,E1 -22040.576,E2 -22040.576} C_VEL
LIN {X 0,Y 189.714,Z 553.16,A -85,B 0,C 180,E1 -22042.298,E2 -22042.298} C_VEL
LIN {X 0,Y 186.537,Z 554.452,A -85,B 0,C 180,E1 -22045.133,E2 -22045.133} C_VEL
LIN {X 0,Y 184.051,Z 555.058,A -85,B 0,C 180,E1 -22047.477,E2 -22047.477} C_VEL
LIN {X 0,Y 183.088,Z 555.239,A -85,B 0,C 180,E1 -22049.311,E2 -22049.311} C_VEL
LIN {X 0,Y 183.056,Z 555.275,A -85,B 0,C 180,E1 -22049.932,E2 -22049.932} C_VEL
LIN {X 0,Y 183.018,Z 554.602,A -85,B 0,C 180,E1 -22054.405,E2 -22054.405} C_VEL
LIN {X 0,Y 183.497,Z 552.58,A -85,B 0,C 180,E1 -22058.812,E2 -22058.812} C_VEL
LIN {X 0,Y 184.627,Z 549.166,A -85,B 0,C 180,E1 -22063.202,E2 -22063.202} C_VEL
LIN {X 0,Y 186.68,Z 544.26,A -85,B 0,C 180,E1 -22067.528,E2 -22067.528} C_VEL
LIN {X 0,Y 189.585,Z 537.717,A -85,B 0,C 180,E1 -22071.759,E2 -22071.759} C_VEL
LIN {X 0,Y 192.806,Z 530.436,A -85,B 0,C 180,E1 -22075.36,E2 -22075.36} C_VEL
LIN {X 0,Y 196.872,Z 521.417,A -85,B 0,C 180,E1 -22078.811,E2 -22078.811} C_VEL
LIN {X 0,Y 200.858,Z 511.956,A -85,B 0,C 180,E1 -22081.658,E2 -22081.658} C_VEL
LIN {X 0,Y 205.213,Z 500.98,A -85,B 0,C 180,E1 -22084.25,E2 -22084.25} C_VEL
LIN {X 0,Y 206.5,Z 497.238,A -85,B 0,C 180,E1 -22085.033,E2 -22085.033} C_VEL
LIN {X 0,Y 206.715,Z 488.591,A -85,B 0,C 180,E1 -22087.119,E2 -22087.119} C_VEL
LIN {X 0,Y 206.2,Z 477.881,A -85,B 0,C 180,E1 -22089.545,E2 -22089.545} C_VEL
LIN {X 0,Y 204.619,Z 466.726,A -85,B 0,C 180,E1 -22091.99,E2 -22091.99} C_VEL
LIN {X 0,Y 202.598,Z 457.835,A -85,B 0,C 180,E1 -22093.93,E2 -22093.93} C_VEL
LIN {X 0,Y 199.645,Z 449.347,A -85,B 0,C 180,E1 -22095.953,E2 -22095.953} C_VEL
LIN {X 0,Y 196.391,Z 442.456,A -85,B 0,C 180,E1 -22097.787,E2 -22097.787} C_VEL
LIN {X 0,Y 194.737,Z 439.194,A -85,B 0,C 180,E1 -22098.672,E2 -22098.672} C_VEL
LIN {X 0,Y 192.392,Z 434.835,A -85,B 0,C 180,E1 -22099.923,E2 -22099.923} C_VEL
LIN {X 0,Y 190.248,Z 431.348,A -85,B 0,C 180,E1 -22101.013,E2 -22101.013} C_VEL
LIN {X 0,Y 189.5,Z 429.774,A -85,B 0,C 180,E1 -22101.439,E2 -22101.439} C_VEL
LIN {X 0,Y 187.36,Z 427.261,A -85,B 0,C 180,E1 -22102.46,E2 -22102.46} C_VEL
LIN {X 0,Y 186.255,Z 424.198,A -85,B 0,C 180,E1 -22103.201,E2 -22103.201} C_VEL
LIN {X 0,Y 185.856,Z 421.96,A -85,B 0,C 180,E1 -22108.035,E2 -22108.035} C_VEL
LIN {X 0,Y 185.559,Z 419.997,A -85,B 0,C 180,E1 -22112.968,E2 -22112.968} C_VEL
LIN {X 0,Y 185.582,Z 419.994,A -85,B 0,C 180,E1 -22117.747,E2 -22117.747} C_VEL
LIN {X 0,Y 185.691,Z 419.975,A -85,B 0,C 180,E1 -22122.375,E2 -22122.375} C_VEL
LIN {X 0,Y 185.766,Z 419.97,A -85,B 0,C 180,E1 -22126.88,E2 -22126.88} C_VEL
LIN {X 0,Y 186.031,Z 419.937,A -85,B 0,C 180,E1 -22131.309,E2 -22131.309} C_VEL
LIN {X 0,Y 186.21,Z 419.914,A -85,B 0,C 180,E1 -22137.837,E2 -22137.837} C_VEL
LIN {X 0,Y 186.411,Z 419.889,A -85,B 0,C 180,E1 -22140,E2 -22140} C_VEL
LIN {X 0,Y 185.929,Z 419.949,A -85,B 0,C 180,E1 -22144.336,E2 -22144.336} C_VEL
LIN {X 0,Y 186.031,Z 419.936,A -85,B 0,C 180,E1 -22148.692,E2 -22148.692} C_VEL
LIN {X 0,Y 185.766,Z 419.964,A -85,B 0,C 180,E1 -22153.12,E2 -22153.12} C_VEL
LIN {X 0,Y 185.692,Z 419.974,A -85,B 0,C 180,E1 -22157.625,E2 -22157.625} C_VEL
LIN {X 0,Y 185.598,Z 419.992,A -85,B 0,C 180,E1 -22162.251,E2 -22162.251} C_VEL
LIN {X 0,Y 185.562,Z 419.996,A -85,B 0,C 180,E1 -22167.032,E2 -22167.032} C_VEL
LIN {X 0,Y 185.578,Z 419.994,A -85,B 0,C 180,E1 -22169.493,E2 -22169.493} C_VEL
LIN {X 0,Y 185.569,Z 420.267,A -85,B 0,C 180,E1 -22172.02,E2 -22172.02} C_VEL
LIN {X 0,Y 185.919,Z 422.259,A -85,B 0,C 180,E1 -22176.793,E2 -22176.793} C_VEL
LIN {X 0,Y 187.033,Z 425.183,A -85,B 0,C 180,E1 -22177.465,E2 -22177.465} C_VEL
LIN {X 0,Y 189.488,Z 428.129,A -85,B 0,C 180,E1 -22178.662,E2 -22178.662} C_VEL
LIN {X 0,Y 191.4,Z 431.71,A -85,B 0,C 180,E1 -22179.701,E2 -22179.701} C_VEL
LIN {X 0,Y 192.915,Z 434.044,A -85,B 0,C 180,E1 -22180.46,E2 -22180.46} C_VEL
LIN {X 0,Y 195.769,Z 439.233,A -85,B 0,C 180,E1 -22181.985,E2 -22181.985} C_VEL
LIN {X 0,Y 199.519,Z 446.864,A -85,B 0,C 180,E1 -22184.082,E2 -22184.082} C_VEL
LIN {X 0,Y 203.194,Z 457.002,A -85,B 0,C 180,E1 -22186.581,E2 -22186.581} C_VEL
LIN {X 0,Y 205.529,Z 466.676,A -85,B 0,C 180,E1 -22188.789,E2 -22188.789} C_VEL
LIN {X 0,Y 207.115,Z 477.744,A -85,B 0,C 180,E1 -22191.303,E2 -22191.303} C_VEL
LIN {X 0,Y 207.573,Z 487.765,A -85,B 0,C 180,E1 -22193.666,E2 -22193.666} C_VEL
LIN {X 0,Y 207.391,Z 492.528,A -85,B 0,C 180,E1 -22194.824,E2 -22194.824} C_VEL
LIN {X 0,Y 203.533,Z 503.025,A -85,B 0,C 180,E1 -22197.054,E2 -22197.054} C_VEL
LIN {X 0,Y 199.956,Z 511.826,A -85,B 0,C 180,E1 -22199.36,E2 -22199.36} C_VEL
LIN {X 0,Y 196.141,Z 520.696,A -85,B 0,C 180,E1 -22202.238,E2 -22202.238} C_VEL
LIN {X 0,Y 192.264,Z 529.19,A -85,B 0,C 180,E1 -22205.718,E2 -22205.718} C_VEL
LIN {X 0,Y 189.274,Z 536.027,A -85,B 0,C 180,E1 -22209.345,E2 -22209.345} C_VEL
LIN {X 0,Y 187.046,Z 540.746,A -85,B 0,C 180,E1 -22212.507,E2 -22212.507} C_VEL
LIN {X 0,Y 184.934,Z 545.633,A -85,B 0,C 180,E1 -22216.82,E2 -22216.82} C_VEL
LIN {X 0,Y 183.722,Z 549.03,A -85,B 0,C 180,E1 -22221.199,E2 -22221.199} C_VEL
LIN {X 0,Y 183.124,Z 551.044,A -85,B 0,C 180,E1 -22225.598,E2 -22225.598} C_VEL
LIN {X 0,Y 183.07,Z 551.728,A -85,B 0,C 180,E1 -22230,E2 -22230} C_VEL
LIN {X 0,Y 183.124,Z 551.094,A -85,B 0,C 180,E1 -22234.402,E2 -22234.402} C_VEL
LIN {X 0,Y 183.693,Z 549.124,A -85,B 0,C 180,E1 -22238.803,E2 -22238.803} C_VEL
LIN {X 0,Y 184.897,Z 545.773,A -85,B 0,C 180,E1 -22243.183,E2 -22243.183} C_VEL
LIN {X 0,Y 187.02,Z 540.938,A -85,B 0,C 180,E1 -22247.496,E2 -22247.496} C_VEL
LIN {X 0,Y 189.211,Z 536.271,A -85,B 0,C 180,E1 -22250.663,E2 -22250.663} C_VEL
LIN {X 0,Y 192.248,Z 529.486,A -85,B 0,C 180,E1 -22254.285,E2 -22254.285} C_VEL
LIN {X 0,Y 195.493,Z 522.406,A -85,B 0,C 180,E1 -22257.282,E2 -22257.282} C_VEL
LIN {X 0,Y 199.256,Z 513.878,A -85,B 0,C 180,E1 -22260.173,E2 -22260.173} C_VEL
LIN {X 0,Y 203.479,Z 503.54,A -85,B 0,C 180,E1 -22262.956,E2 -22262.956} C_VEL
LIN {X 0,Y 207.306,Z 493.148,A -85,B 0,C 180,E1 -22265.193,E2 -22265.193} C_VEL
LIN {X 0,Y 207.668,Z 490.931,A -85,B 0,C 180,E1 -22265.686,E2 -22265.686} C_VEL
LIN {X 0,Y 207.356,Z 479.883,A -85,B 0,C 180,E1 -22268.338,E2 -22268.338} C_VEL
LIN {X 0,Y 205.909,Z 468.44,A -85,B 0,C 180,E1 -22270.96,E2 -22270.96} C_VEL
LIN {X 0,Y 203.371,Z 457.497,A -85,B 0,C 180,E1 -22273.472,E2 -22273.472} C_VEL
LIN {X 0,Y 200.516,Z 449.118,A -85,B 0,C 180,E1 -22275.493,E2 -22275.493} C_VEL
LIN {X 0,Y 196.387,Z 440.414,A -85,B 0,C 180,E1 -22277.874,E2 -22277.874} C_VEL
LIN {X 0,Y 194.392,Z 436.771,A -85,B 0,C 180,E1 -22278.93,E2 -22278.93} C_VEL
LIN {X 0,Y 191.927,Z 432.367,A -85,B 0,C 180,E1 -22280.25,E2 -22280.25} C_VEL
LIN {X 0,Y 189.832,Z 428.957,A -85,B 0,C 180,E1 -22281.335,E2 -22281.335} C_VEL
LIN {X 0,Y 189.211,Z 427.656,A -85,B 0,C 180,E1 -22281.694,E2 -22281.694} C_VEL
LIN {X 0,Y 186.979,Z 425.088,A -85,B 0,C 180,E1 -22282.776,E2 -22282.776} C_VEL
LIN {X 0,Y 185.902,Z 422.175,A -85,B 0,C 180,E1 -22283.457,E2 -22283.457} C_VEL
LIN {X 0,Y 185.572,Z 420.363,A -85,B 0,C 180,E1 -22287.98,E2 -22287.98} C_VEL
LIN {X 0,Y 185.584,Z 419.989,A -85,B 0,C 180,E1 -22290.576,E2 -22290.576} C_VEL
LIN {X 0,Y 185.59,Z 419.989,A -85,B 0,C 180,E1 -22295.383,E2 -22295.383} C_VEL
LIN {X 0,Y 185.61,Z 419.983,A -85,B 0,C 180,E1 -22300.075,E2 -22300.075} C_VEL
LIN {X 0,Y 185.703,Z 419.977,A -85,B 0,C 180,E1 -22304.638,E2 -22304.638} C_VEL
LIN {X 0,Y 185.945,Z 419.947,A -85,B 0,C 180,E1 -22309.328,E2 -22309.328} C_VEL
LIN {X 0,Y 185.972,Z 419.943,A -85,B 0,C 180,E1 -22313.49,E2 -22313.49} C_VEL
LIN {X 0,Y 186.211,Z 419.914,A -85,B 0,C 180,E1 -22317.837,E2 -22317.837} C_VEL
LIN {X 0,Y 186.41,Z 419.89,A -85,B 0,C 180,E1 -22320,E2 -22320} C_VEL
LIN {X 0,Y 185.931,Z 419.95,A -85,B 0,C 180,E1 -22324.335,E2 -22324.335} C_VEL
LIN {X 0,Y 186.032,Z 419.937,A -85,B 0,C 180,E1 -22328.691,E2 -22328.691} C_VEL
LIN {X 0,Y 185.768,Z 419.97,A -85,B 0,C 180,E1 -22333.12,E2 -22333.12} C_VEL
LIN {X 0,Y 185.693,Z 419.979,A -85,B 0,C 180,E1 -22337.624,E2 -22337.624} C_VEL
LIN {X 0,Y 185.599,Z 419.992,A -85,B 0,C 180,E1 -22342.251,E2 -22342.251} C_VEL
LIN {X 0,Y 185.565,Z 420.016,A -85,B 0,C 180,E1 -22347.032,E2 -22347.032} C_VEL
LIN {X 0,Y 185.766,Z 420.974,A -85,B 0,C 180,E1 -22349.523,E2 -22349.523} C_VEL
LIN {X 0,Y 186.032,Z 423.17,A -85,B 0,C 180,E1 -22354.519,E2 -22354.519} C_VEL
LIN {X 0,Y 186.241,Z 424.214,A -85,B 0,C 180,E1 -22356.718,E2 -22356.718} C_VEL
LIN {X 0,Y 187.45,Z 427.409,A -85,B 0,C 180,E1 -22357.466,E2 -22357.466} C_VEL
LIN {X 0,Y 189.879,Z 430.364,A -85,B 0,C 180,E1 -22358.645,E2 -22358.645} C_VEL
LIN {X 0,Y 191.812,Z 434.098,A -85,B 0,C 180,E1 -22359.696,E2 -22359.696} C_VEL
LIN {X 0,Y 193.192,Z 436.131,A -85,B 0,C 180,E1 -22360.369,E2 -22360.369} C_VEL
LIN {X 0,Y 195.993,Z 441.54,A -85,B 0,C 180,E1 -22361.888,E2 -22361.888} C_VEL
LIN {X 0,Y 198.953,Z 447.625,A -85,B 0,C 180,E1 -22363.538,E2 -22363.538} C_VEL
LIN {X 0,Y 202.143,Z 456.143,A -85,B 0,C 180,E1 -22365.6,E2 -22365.6} C_VEL
LIN {X 0,Y 204.073,Z 463.708,A -85,B 0,C 180,E1 -22367.287,E2 -22367.287} C_VEL
LIN {X 0,Y 205.621,Z 472.451,A -85,B 0,C 180,E1 -22369.197,E2 -22369.197} C_VEL
LIN {X 0,Y 206.676,Z 482.553,A -85,B 0,C 180,E1 -22371.454,E2 -22371.454} C_VEL
LIN {X 0,Y 206.749,Z 493.892,A -85,B 0,C 180,E1 -22374.099,E2 -22374.099} C_VEL
LIN {X 0,Y 206.517,Z 497.401,A -85,B 0,C 180,E1 -22374.945,E2 -22374.945} C_VEL
LIN {X 0,Y 202.317,Z 508.587,A -85,B 0,C 180,E1 -22377.423,E2 -22377.423} C_VEL
LIN {X 0,Y 198.099,Z 518.606,A -85,B 0,C 180,E1 -22380.219,E2 -22380.219} C_VEL
LIN {X 0,Y 194.485,Z 526.928,A -85,B 0,C 180,E1 -22383.147,E2 -22383.147} C_VEL
LIN {X 0,Y 190.789,Z 534.985,A -85,B 0,C 180,E1 -22386.729,E2 -22386.729} C_VEL
LIN {X 0,Y 187.995,Z 541.293,A -85,B 0,C 180,E1 -22390.339,E2 -22390.339} C_VEL
LIN {X 0,Y 186.062,Z 545.729,A -85,B 0,C 180,E1 -22393.543,E2 -22393.543} C_VEL
LIN {X 0,Y 184.633,Z 549.22,A -85,B 0,C 180,E1 -22396.798,E2 -22396.798} C_VEL
LIN {X 0,Y 183.492,Z 552.614,A -85,B 0,C 180,E1 -22401.187,E2 -22401.187} C_VEL
LIN {X 0,Y 183.017,Z 554.62,A -85,B 0,C 180,E1 -22405.595,E2 -22405.595} C_VEL
LIN {X 0,Y 183.056,Z 555.275,A -85,B 0,C 180,E1 -22409.932,E2 -22409.932} C_VEL
LIN {X 0,Y 182.494,Z 555.26,A -85,B 0,C 180,E1 -22411.768,E2 -22411.768} C_VEL
LIN {X 0,Y 180.95,Z 554.967,A -85,B 0,C 180,E1 -22413.574,E2 -22413.574} C_VEL
LIN {X 0,Y 177.358,Z 553.6,A -85,B 0,C 180,E1 -22417.218,E2 -22417.218} C_VEL
LIN {X 0,Y 176.529,Z 552.546,A -85,B 0,C 180,E1 -22419.107,E2 -22419.107} C_VEL
LIN {X 0,Y 176.556,Z 552.127,A -85,B 0,C 180,E1 -22419.741,E2 -22419.741} C_VEL
LIN {X 0,Y 177.688,Z 549.096,A -85,B 0,C 180,E1 -22423.728,E2 -22423.728} C_VEL
LIN {X 0,Y 179.893,Z 544.19,A -85,B 0,C 180,E1 -22428.212,E2 -22428.212} C_VEL
LIN {X 0,Y 182.924,Z 537.646,A -85,B 0,C 180,E1 -22432.594,E2 -22432.594} C_VEL
LIN {X 0,Y 186.368,Z 530.365,A -85,B 0,C 180,E1 -22436.301,E2 -22436.301} C_VEL
LIN {X 0,Y 190.664,Z 521.346,A -85,B 0,C 180,E1 -22439.842,E2 -22439.842} C_VEL
LIN {X 0,Y 194.829,Z 511.884,A -85,B 0,C 180,E1 -22442.758,E2 -22442.758} C_VEL
LIN {X 0,Y 199.172,Z 501.449,A -85,B 0,C 180,E1 -22445.285,E2 -22445.285} C_VEL
LIN {X 0,Y 200.28,Z 498.278,A -85,B 0,C 180,E1 -22445.975,E2 -22445.975} C_VEL
LIN {X 0,Y 200.583,Z 487.626,A -85,B 0,C 180,E1 -22448.675,E2 -22448.675} C_VEL
LIN {X 0,Y 200.081,Z 478.031,A -85,B 0,C 180,E1 -22450.959,E2 -22450.959} C_VEL
LIN {X 0,Y 198.771,Z 468.109,A -85,B 0,C 180,E1 -22453.269,E2 -22453.269} C_VEL
LIN {X 0,Y 196.912,Z 459.854,A -85,B 0,C 180,E1 -22455.209,E2 -22455.209} C_VEL
LIN {X 0,Y 194.158,Z 451.97,A -85,B 0,C 180,E1 -22457.258,E2 -22457.258} C_VEL
LIN {X 0,Y 190.231,Z 443.56,A -85,B 0,C 180,E1 -22459.72,E2 -22459.72} C_VEL
LIN {X 0,Y 188.271,Z 439.832,A -85,B 0,C 180,E1 -22460.875,E2 -22460.875} C_VEL
LIN {X 0,Y 186.104,Z 435.662,A -85,B 0,C 180,E1 -22462.19,E2 -22462.19} C_VEL
LIN {X 0,Y 183.642,Z 432.208,A -85,B 0,C 180,E1 -22463.535,E2 -22463.535} C_VEL
LIN {X 0,Y 182.46,Z 429.789,A -85,B 0,C 180,E1 -22464.287,E2 -22464.287} C_VEL
LIN {X 0,Y 180.144,Z 427.084,A -85,B 0,C 180,E1 -22465.559,E2 -22465.559} C_VEL
LIN {X 0,Y 179.015,Z 424.07,A -85,B 0,C 180,E1 -22466.434,E2 -22466.434} C_VEL
LIN {X 0,Y 178.656,Z 421.876,A -85,B 0,C 180,E1 -22471.832,E2 -22471.832} C_VEL
LIN {X 0,Y 178.514,Z 420.875,A -85,B 0,C 180,E1 -22474.89,E2 -22474.89} C_VEL
LIN {X 0,Y 178.623,Z 420.861,A -85,B 0,C 180,E1 -22480.785,E2 -22480.785} C_VEL
LIN {X 0,Y 178.667,Z 420.855,A -85,B 0,C 180,E1 -22484.017,E2 -22484.017} C_VEL
LIN {X 0,Y 178.896,Z 420.819,A -85,B 0,C 180,E1 -22489.153,E2 -22489.153} C_VEL
LIN {X 0,Y 178.936,Z 420.813,A -85,B 0,C 180,E1 -22493.233,E2 -22493.233} C_VEL
LIN {X 0,Y 179.156,Z 420.792,A -85,B 0,C 180,E1 -22497.752,E2 -22497.752} C_VEL
LIN {X 0,Y 179.374,Z 420.765,A -85,B 0,C 180,E1 -22500,E2 -22500} C_VEL
LIN {X 0,Y 178.877,Z 420.827,A -85,B 0,C 180,E1 -22504.507,E2 -22504.507} C_VEL
LIN {X 0,Y 178.98,Z 420.815,A -85,B 0,C 180,E1 -22509.037,E2 -22509.037} C_VEL
LIN {X 0,Y 178.689,Z 420.844,A -85,B 0,C 180,E1 -22513.65,E2 -22513.65} C_VEL
LIN {X 0,Y 178.651,Z 420.855,A -85,B 0,C 180,E1 -22518.344,E2 -22518.344} C_VEL
LIN {X 0,Y 178.512,Z 420.874,A -85,B 0,C 180,E1 -22523.185,E2 -22523.185} C_VEL
LIN {X 0,Y 178.487,Z 420.877,A -85,B 0,C 180,E1 -22528.197,E2 -22528.197} C_VEL
LIN {X 0,Y 178.55,Z 421.283,A -85,B 0,C 180,E1 -22530.777,E2 -22530.777} C_VEL
LIN {X 0,Y 178.711,Z 422.337,A -85,B 0,C 180,E1 -22533.574,E2 -22533.574} C_VEL
LIN {X 0,Y 179.831,Z 425.188,A -85,B 0,C 180,E1 -22534.347,E2 -22534.347} C_VEL
LIN {X 0,Y 182.226,Z 427.865,A -85,B 0,C 180,E1 -22535.67,E2 -22535.67} C_VEL
LIN {X 0,Y 184.669,Z 432.22,A -85,B 0,C 180,E1 -22537.153,E2 -22537.153} C_VEL
LIN {X 0,Y 185.999,Z 434.055,A -85,B 0,C 180,E1 -22537.88,E2 -22537.88} C_VEL
LIN {X 0,Y 188.287,Z 438.01,A -85,B 0,C 180,E1 -22539.232,E2 -22539.232} C_VEL
LIN {X 0,Y 191.991,Z 445.248,A -85,B 0,C 180,E1 -22541.479,E2 -22541.479} C_VEL
LIN {X 0,Y 195.465,Z 453.06,A -85,B 0,C 180,E1 -22543.733,E2 -22543.733} C_VEL
LIN {X 0,Y 198.024,Z 461.061,A -85,B 0,C 180,E1 -22545.816,E2 -22545.816} C_VEL
LIN {X 0,Y 200.025,Z 470.513,A -85,B 0,C 180,E1 -22548.12,E2 -22548.12} C_VEL
LIN {X 0,Y 201.221,Z 481.399,A -85,B 0,C 180,E1 -22550.764,E2 -22550.764} C_VEL
LIN {X 0,Y 201.365,Z 491.805,A -85,B 0,C 180,E1 -22553.393,E2 -22553.393} C_VEL
LIN {X 0,Y 201.047,Z 494.277,A -85,B 0,C 180,E1 -22553.986,E2 -22553.986} C_VEL
LIN {X 0,Y 196.821,Z 505.012,A -85,B 0,C 180,E1 -22556.395,E2 -22556.395} C_VEL
LIN {X 0,Y 192.479,Z 515.057,A -85,B 0,C 180,E1 -22559.258,E2 -22559.258} C_VEL
LIN {X 0,Y 188.596,Z 523.398,A -85,B 0,C 180,E1 -22562.237,E2 -22562.237} C_VEL
LIN {X 0,Y 185.25,Z 530.357,A -85,B 0,C 180,E1 -22565.335,E2 -22565.335} C_VEL
LIN {X 0,Y 182.59,Z 536.098,A -85,B 0,C 180,E1 -22568.552,E2 -22568.552} C_VEL
LIN {X 0,Y 180.279,Z 540.816,A -85,B 0,C 180,E1 -22571.828,E2 -22571.828} C_VEL
LIN {X 0,Y 178,Z 545.703,A -85,B 0,C 180,E1 -22576.297,E2 -22576.297} C_VEL
LIN {X 0,Y 176.676,Z 549.1,A -85,B 0,C 180,E1 -22580.845,E2 -22580.845} C_VEL
LIN {X 0,Y 176.035,Z 551.113,A -85,B 0,C 180,E1 -22585.42,E2 -22585.42} C_VEL
LIN {X 0,Y 175.983,Z 551.797,A -85,B 0,C 180,E1 -22590,E2 -22590} C_VEL
LIN {X 0,Y 176.035,Z 551.162,A -85,B 0,C 180,E1 -22594.58,E2 -22594.58} C_VEL
LIN {X 0,Y 176.317,Z 550.346,A -85,B 0,C 180,E1 -22596.868,E2 -22596.868} C_VEL
LIN {X 0,Y 177.208,Z 547.694,A -85,B 0,C 180,E1 -22601.438,E2 -22601.438} C_VEL
LIN {X 0,Y 178.93,Z 543.618,A -85,B 0,C 180,E1 -22605.959,E2 -22605.959} C_VEL
LIN {X 0,Y 181.77,Z 537.985,A -85,B 0,C 180,E1 -22610.364,E2 -22610.364} C_VEL
LIN {X 0,Y 184.595,Z 531.944,A -85,B 0,C 180,E1 -22613.972,E2 -22613.972} C_VEL
LIN {X 0,Y 187.961,Z 524.949,A -85,B 0,C 180,E1 -22617.261,E2 -22617.261} C_VEL
LIN {X 0,Y 191.717,Z 516.929,A -85,B 0,C 180,E1 -22620.269,E2 -22620.269} C_VEL
LIN {X 0,Y 196.048,Z 507.254,A -85,B 0,C 180,E1 -22623.14,E2 -22623.14} C_VEL
LIN {X 0,Y 200.454,Z 496.185,A -85,B 0,C 180,E1 -22625.75,E2 -22625.75} C_VEL
LIN {X 0,Y 201.428,Z 493.214,A -85,B 0,C 180,E1 -22626.381,E2 -22626.381} C_VEL
LIN {X 0,Y 201.373,Z 482.413,A -85,B 0,C 180,E1 -22629.136,E2 -22629.136} C_VEL
LIN {X 0,Y 200.083,Z 470.403,A -85,B 0,C 180,E1 -22632.059,E2 -22632.059} C_VEL
LIN {X 0,Y 197.994,Z 460.812,A -85,B 0,C 180,E1 -22634.418,E2 -22634.418} C_VEL
LIN {X 0,Y 195,Z 451.83,A -85,B 0,C 180,E1 -22636.781,E2 -22636.781} C_VEL
LIN {X 0,Y 190.796,Z 442.675,A -85,B 0,C 180,E1 -22639.473,E2 -22639.473} C_VEL
LIN {X 0,Y 187.866,Z 437.382,A -85,B 0,C 180,E1 -22641.207,E2 -22641.207} C_VEL
LIN {X 0,Y 185.316,Z 432.94,A -85,B 0,C 180,E1 -22642.726,E2 -22642.726} C_VEL
LIN {X 0,Y 183.073,Z 429.589,A -85,B 0,C 180,E1 -22644.005,E2 -22644.005} C_VEL
LIN {X 0,Y 182.216,Z 427.867,A -85,B 0,C 180,E1 -22644.558,E2 -22644.558} C_VEL
LIN {X 0,Y 179.972,Z 425.43,A -85,B 0,C 180,E1 -22645.799,E2 -22645.799} C_VEL
LIN {X 0,Y 178.72,Z 422.259,A -85,B 0,C 180,E1 -22646.764,E2 -22646.764} C_VEL
LIN {X 0,Y 178.528,Z 421.104,A -85,B 0,C 180,E1 -22650.005,E2 -22650.005} C_VEL
LIN {X 0,Y 178.537,Z 420.872,A -85,B 0,C 180,E1 -22654.876,E2 -22654.876} C_VEL
LIN {X 0,Y 178.626,Z 420.857,A -85,B 0,C 180,E1 -22660.784,E2 -22660.784} C_VEL
LIN {X 0,Y 178.684,Z 420.851,A -85,B 0,C 180,E1 -22666.35,E2 -22666.35} C_VEL
LIN {X 0,Y 178.981,Z 420.813,A -85,B 0,C 180,E1 -22670.963,E2 -22670.963} C_VEL
LIN {X 0,Y 179.157,Z 420.793,A -85,B 0,C 180,E1 -22677.752,E2 -22677.752} C_VEL
LIN {X 0,Y 179.373,Z 420.767,A -85,B 0,C 180,E1 -22680,E2 -22680} C_VEL
LIN {X 0,Y 178.88,Z 420.829,A -85,B 0,C 180,E1 -22684.507,E2 -22684.507} C_VEL
LIN {X 0,Y 178.981,Z 420.816,A -85,B 0,C 180,E1 -22689.037,E2 -22689.037} C_VEL
LIN {X 0,Y 178.69,Z 420.853,A -85,B 0,C 180,E1 -22693.649,E2 -22693.649} C_VEL
LIN {X 0,Y 178.652,Z 420.857,A -85,B 0,C 180,E1 -22698.343,E2 -22698.343} C_VEL
LIN {X 0,Y 178.513,Z 420.867,A -85,B 0,C 180,E1 -22703.185,E2 -22703.185} C_VEL
LIN {X 0,Y 178.539,Z 421.032,A -85,B 0,C 180,E1 -22705.658,E2 -22705.658} C_VEL
LIN {X 0,Y 178.827,Z 422.924,A -85,B 0,C 180,E1 -22710.724,E2 -22710.724} C_VEL
LIN {X 0,Y 179.058,Z 424.327,A -85,B 0,C 180,E1 -22713.557,E2 -22713.557} C_VEL
LIN {X 0,Y 180.239,Z 427.243,A -85,B 0,C 180,E1 -22714.358,E2 -22714.358} C_VEL
LIN {X 0,Y 182.941,Z 430.508,A -85,B 0,C 180,E1 -22715.864,E2 -22715.864} C_VEL
LIN {X 0,Y 184.877,Z 434.205,A -85,B 0,C 180,E1 -22717.05,E2 -22717.05} C_VEL
LIN {X 0,Y 186.338,Z 436.16,A -85,B 0,C 180,E1 -22717.835,E2 -22717.835} C_VEL
LIN {X 0,Y 188.537,Z 440.165,A -85,B 0,C 180,E1 -22719.147,E2 -22719.147} C_VEL
LIN {X 0,Y 191.672,Z 446.43,A -85,B 0,C 180,E1 -22721.052,E2 -22721.052} C_VEL
LIN {X 0,Y 195.792,Z 456.13,A -85,B 0,C 180,E1 -22723.761,E2 -22723.761} C_VEL
LIN {X 0,Y 198.169,Z 464.592,A -85,B 0,C 180,E1 -22725.86,E2 -22725.86} C_VEL
LIN {X 0,Y 199.882,Z 475.338,A -85,B 0,C 180,E1 -22728.344,E2 -22728.344} C_VEL
LIN {X 0,Y 200.677,Z 484.949,A -85,B 0,C 180,E1 -22730.637,E2 -22730.637} C_VEL
LIN {X 0,Y 200.494,Z 496.18,A -85,B 0,C 180,E1 -22733.422,E2 -22733.422} C_VEL
LIN {X 0,Y 200.327,Z 498.431,A -85,B 0,C 180,E1 -22734.007,E2 -22734.007} C_VEL
LIN {X 0,Y 196.355,Z 508.52,A -85,B 0,C 180,E1 -22736.304,E2 -22736.304} C_VEL
LIN {X 0,Y 191.93,Z 518.539,A -85,B 0,C 180,E1 -22739.159,E2 -22739.159} C_VEL
LIN {X 0,Y 188.139,Z 526.861,A -85,B 0,C 180,E1 -22742.164,E2 -22742.164} C_VEL
LIN {X 0,Y 184.251,Z 534.919,A -85,B 0,C 180,E1 -22745.852,E2 -22745.852} C_VEL
LIN {X 0,Y 182.075,Z 539.561,A -85,B 0,C 180,E1 -22748.488,E2 -22748.488} C_VEL
LIN {X 0,Y 179.892,Z 544.271,A -85,B 0,C 180,E1 -22751.787,E2 -22751.787} C_VEL
LIN {X 0,Y 177.693,Z 549.152,A -85,B 0,C 180,E1 -22756.272,E2 -22756.272} C_VEL
LIN {X 0,Y 176.452,Z 552.546,A -85,B 0,C 180,E1 -22760.832,E2 -22760.832} C_VEL
LIN {X 0,Y 175.94,Z 554.552,A -85,B 0,C 180,E1 -22765.417,E2 -22765.417} C_VEL
LIN {X 0,Y 175.974,Z 555.212,A -85,B 0,C 180,E1 -22770,E2 -22770} C_VEL
LIN {X 0,Y 175.941,Z 554.532,A -85,B 0,C 180,E1 -22774.582,E2 -22774.582} C_VEL
LIN {X 0,Y 176.456,Z 552.51,A -85,B 0,C 180,E1 -22779.167,E2 -22779.167} C_VEL
LIN {X 0,Y 176.556,Z 552.127,A -85,B 0,C 180,E1 -22779.741,E2 -22779.741} C_VEL
LIN {X 0,Y 176.332,Z 550.897,A -85,B 0,C 180,E1 -22781.608,E2 -22781.608} C_VEL
LIN {X 0,Y 174.536,Z 548.426,A -85,B 0,C 180,E1 -22784.689,E2 -22784.689} C_VEL
LIN {X 0,Y 173.262,Z 546.095,A -85,B 0,C 180,E1 -22787.161,E2 -22787.161} C_VEL
LIN {X 0,Y 173.244,Z 544.049,A -85,B 0,C 180,E1 -22789.002,E2 -22789.002} C_VEL
LIN {X 0,Y 173.526,Z 543.303,A -85,B 0,C 180,E1 -22789.602,E2 -22789.602} C_VEL
LIN {X 0,Y 176.403,Z 537.391,A -85,B 0,C 180,E1 -22793.604,E2 -22793.604} C_VEL
LIN {X 0,Y 179.984,Z 530.294,A -85,B 0,C 180,E1 -22797.31,E2 -22797.31} C_VEL
LIN {X 0,Y 184.522,Z 521.274,A -85,B 0,C 180,E1 -22800.943,E2 -22800.943} C_VEL
LIN {X 0,Y 188.885,Z 511.812,A -85,B 0,C 180,E1 -22803.925,E2 -22803.925} C_VEL
LIN {X 0,Y 193.731,Z 500.468,A -85,B 0,C 180,E1 -22806.706,E2 -22806.706} C_VEL
LIN {X 0,Y 194.282,Z 497.171,A -85,B 0,C 180,E1 -22807.576,E2 -22807.576} C_VEL
LIN {X 0,Y 194.528,Z 485.789,A -85,B 0,C 180,E1 -22810.565,E2 -22810.565} C_VEL
LIN {X 0,Y 193.655,Z 474.19,A -85,B 0,C 180,E1 -22813.463,E2 -22813.463} C_VEL
LIN {X 0,Y 192.251,Z 465.85,A -85,B 0,C 180,E1 -22815.531,E2 -22815.531} C_VEL
LIN {X 0,Y 189.452,Z 456.425,A -85,B 0,C 180,E1 -22818.107,E2 -22818.107} C_VEL
LIN {X 0,Y 184.718,Z 445.684,A -85,B 0,C 180,E1 -22821.463,E2 -22821.463} C_VEL
LIN {X 0,Y 182.412,Z 441.258,A -85,B 0,C 180,E1 -22823.004,E2 -22823.004} C_VEL
LIN {X 0,Y 179.825,Z 436.993,A -85,B 0,C 180,E1 -22824.664,E2 -22824.664} C_VEL
LIN {X 0,Y 179.051,Z 435.458,A -85,B 0,C 180,E1 -22825.209,E2 -22825.209} C_VEL
LIN {X 0,Y 176.782,Z 432.361,A -85,B 0,C 180,E1 -22826.627,E2 -22826.627} C_VEL
LIN {X 0,Y 175.641,Z 429.952,A -85,B 0,C 180,E1 -22827.473,E2 -22827.473} C_VEL
LIN {X 0,Y 173.21,Z 427.376,A -85,B 0,C 180,E1 -22829.02,E2 -22829.02} C_VEL
LIN {X 0,Y 171.897,Z 424.324,A -85,B 0,C 180,E1 -22830.049,E2 -22830.049} C_VEL
LIN {X 0,Y 171.802,Z 423.914,A -85,B 0,C 180,E1 -22830.316,E2 -22830.316} C_VEL
LIN {X 0,Y 171.476,Z 422.02,A -85,B 0,C 180,E1 -22835.805,E2 -22835.805} C_VEL
LIN {X 0,Y 171.579,Z 421.738,A -85,B 0,C 180,E1 -22840.872,E2 -22840.872} C_VEL
LIN {X 0,Y 171.61,Z 421.728,A -85,B 0,C 180,E1 -22845.776,E2 -22845.776} C_VEL
LIN {X 0,Y 171.912,Z 421.696,A -85,B 0,C 180,E1 -22850.589,E2 -22850.589} C_VEL
LIN {X 0,Y 171.828,Z 421.706,A -85,B 0,C 180,E1 -22855.308,E2 -22855.308} C_VEL
LIN {X 0,Y 172.336,Z 421.642,A -85,B 0,C 180,E1 -22860,E2 -22860} C_VEL
LIN {X 0,Y 171.827,Z 421.705,A -85,B 0,C 180,E1 -22864.692,E2 -22864.692} C_VEL
LIN {X 0,Y 171.912,Z 421.697,A -85,B 0,C 180,E1 -22869.412,E2 -22869.412} C_VEL
LIN {X 0,Y 171.611,Z 421.727,A -85,B 0,C 180,E1 -22874.225,E2 -22874.225} C_VEL
LIN {X 0,Y 171.546,Z 421.741,A -85,B 0,C 180,E1 -22879.562,E2 -22879.562} C_VEL
LIN {X 0,Y 171.47,Z 421.751,A -85,B 0,C 180,E1 -22885.616,E2 -22885.616} C_VEL
LIN {X 0,Y 171.581,Z 422.462,A -85,B 0,C 180,E1 -22889.793,E2 -22889.793} C_VEL
LIN {X 0,Y 172.753,Z 425.402,A -85,B 0,C 180,E1 -22890.748,E2 -22890.748} C_VEL
LIN {X 0,Y 174.911,Z 427.902,A -85,B 0,C 180,E1 -22892.168,E2 -22892.168} C_VEL
LIN {X 0,Y 175.722,Z 428.692,A -85,B 0,C 180,E1 -22892.681,E2 -22892.681} C_VEL
LIN {X 0,Y 177.418,Z 431.988,A -85,B 0,C 180,E1 -22893.9,E2 -22893.9} C_VEL
LIN {X 0,Y 179.255,Z 434.249,A -85,B 0,C 180,E1 -22895.025,E2 -22895.025} C_VEL
LIN {X 0,Y 181.287,Z 438.005,A -85,B 0,C 180,E1 -22896.42,E2 -22896.42} C_VEL
LIN {X 0,Y 182.628,Z 440.268,A -85,B 0,C 180,E1 -22897.276,E2 -22897.276} C_VEL
LIN {X 0,Y 186.467,Z 447.556,A -85,B 0,C 180,E1 -22899.847,E2 -22899.847} C_VEL
LIN {X 0,Y 190.543,Z 457.307,A -85,B 0,C 180,E1 -22902.884,E2 -22902.884} C_VEL
LIN {X 0,Y 192.901,Z 465.474,A -85,B 0,C 180,E1 -22905.132,E2 -22905.132} C_VEL
LIN {X 0,Y 194.441,Z 474.273,A -85,B 0,C 180,E1 -22907.428,E2 -22907.428} C_VEL
LIN {X 0,Y 195.285,Z 484.846,A -85,B 0,C 180,E1 -22910.166,E2 -22910.166} C_VEL
LIN {X 0,Y 195.154,Z 494.353,A -85,B 0,C 180,E1 -22912.718,E2 -22912.718} C_VEL
LIN {X 0,Y 193.312,Z 499.61,A -85,B 0,C 180,E1 -22913.904,E2 -22913.904} C_VEL
LIN {X 0,Y 188.555,Z 510.346,A -85,B 0,C 180,E1 -22916.648,E2 -22916.648} C_VEL
LIN {X 0,Y 184.322,Z 519.488,A -85,B 0,C 180,E1 -22919.655,E2 -22919.655} C_VEL
LIN {X 0,Y 179.904,Z 528.219,A -85,B 0,C 180,E1 -22923.305,E2 -22923.305} C_VEL
LIN {X 0,Y 176.852,Z 534.366,A -85,B 0,C 180,E1 -22926.585,E2 -22926.585} C_VEL
LIN {X 0,Y 174.309,Z 539.448,A -85,B 0,C 180,E1 -22929.958,E2 -22929.958} C_VEL
LIN {X 0,Y 171.578,Z 544.712,A -85,B 0,C 180,E1 -22934.559,E2 -22934.559} C_VEL
LIN {X 0,Y 170.263,Z 547.65,A -85,B 0,C 180,E1 -22938.09,E2 -22938.09} C_VEL
LIN {X 0,Y 169.261,Z 550.344,A -85,B 0,C 180,E1 -22942.845,E2 -22942.845} C_VEL
LIN {X 0,Y 168.859,Z 551.689,A -85,B 0,C 180,E1 -22947.615,E2 -22947.615} C_VEL
LIN {X 0,Y 168.882,Z 551.865,A -85,B 0,C 180,E1 -22950,E2 -22950} C_VEL
LIN {X 0,Y 168.952,Z 551.231,A -85,B 0,C 180,E1 -22954.772,E2 -22954.772} C_VEL
LIN {X 0,Y 169.634,Z 549.261,A -85,B 0,C 180,E1 -22959.539,E2 -22959.539} C_VEL
LIN {X 0,Y 171.063,Z 545.909,A -85,B 0,C 180,E1 -22964.271,E2 -22964.271} C_VEL
LIN {X 0,Y 173.482,Z 541.074,A -85,B 0,C 180,E1 -22968.911,E2 -22968.911} C_VEL
LIN {X 0,Y 176.853,Z 534.602,A -85,B 0,C 180,E1 -22973.416,E2 -22973.416} C_VEL
LIN {X 0,Y 180.452,Z 527.394,A -85,B 0,C 180,E1 -22977.234,E2 -22977.234} C_VEL
LIN {X 0,Y 184.923,Z 518.474,A -85,B 0,C 180,E1 -22980.869,E2 -22980.869} C_VEL
LIN {X 0,Y 189.311,Z 509.099,A -85,B 0,C 180,E1 -22983.839,E2 -22983.839} C_VEL
LIN {X 0,Y 193.91,Z 498.323,A -85,B 0,C 180,E1 -22986.525,E2 -22986.525} C_VEL
LIN {X 0,Y 195.23,Z 494.725,A -85,B 0,C 180,E1 -22987.323,E2 -22987.323} C_VEL
LIN {X 0,Y 195.404,Z 485.267,A -85,B 0,C 180,E1 -22989.866,E2 -22989.866} C_VEL
LIN {X 0,Y 194.58,Z 474.699,A -85,B 0,C 180,E1 -22992.616,E2 -22992.616} C_VEL
LIN {X 0,Y 192.915,Z 465.256,A -85,B 0,C 180,E1 -22995.091,E2 -22995.091} C_VEL
LIN {X 0,Y 190.75,Z 457.702,A -85,B 0,C 180,E1 -22997.174,E2 -22997.174} C_VEL
LIN {X 0,Y 186.699,Z 447.928,A -85,B 0,C 180,E1 -23000.212,E2 -23000.212} C_VEL
LIN {X 0,Y 183.574,Z 442.06,A -85,B 0,C 180,E1 -23002.29,E2 -23002.29} C_VEL
LIN {X 0,Y 181.577,Z 438.349,A -85,B 0,C 180,E1 -23003.633,E2 -23003.633} C_VEL
LIN {X 0,Y 179.363,Z 434.498,A -85,B 0,C 180,E1 -23005.123,E2 -23005.123} C_VEL
LIN {X 0,Y 178.176,Z 432.925,A -85,B 0,C 180,E1 -23005.869,E2 -23005.869} C_VEL
LIN {X 0,Y 176.135,Z 429.697,A -85,B 0,C 180,E1 -23007.237,E2 -23007.237} C_VEL
LIN {X 0,Y 175.428,Z 428.25,A -85,B 0,C 180,E1 -23007.769,E2 -23007.769} C_VEL
LIN {X 0,Y 172.909,Z 425.652,A -85,B 0,C 180,E1 -23009.4,E2 -23009.4} C_VEL
LIN {X 0,Y 171.601,Z 422.647,A -85,B 0,C 180,E1 -23010.445,E2 -23010.445} C_VEL
LIN {X 0,Y 171.544,Z 422.412,A -85,B 0,C 180,E1 -23010.552,E2 -23010.552} C_VEL
LIN {X 0,Y 171.472,Z 421.751,A -85,B 0,C 180,E1 -23014.383,E2 -23014.383} C_VEL
LIN {X 0,Y 171.582,Z 421.734,A -85,B 0,C 180,E1 -23020.872,E2 -23020.872} C_VEL
LIN {X 0,Y 171.597,Z 421.736,A -85,B 0,C 180,E1 -23025.774,E2 -23025.774} C_VEL
LIN {X 0,Y 171.913,Z 421.695,A -85,B 0,C 180,E1 -23030.588,E2 -23030.588} C_VEL
LIN {X 0,Y 171.828,Z 421.705,A -85,B 0,C 180,E1 -23035.308,E2 -23035.308} C_VEL
LIN {X 0,Y 172.336,Z 421.643,A -85,B 0,C 180,E1 -23040,E2 -23040} C_VEL
LIN {X 0,Y 171.829,Z 421.707,A -85,B 0,C 180,E1 -23044.692,E2 -23044.692} C_VEL
LIN {X 0,Y 171.913,Z 421.697,A -85,B 0,C 180,E1 -23049.411,E2 -23049.411} C_VEL
LIN {X 0,Y 171.612,Z 421.733,A -85,B 0,C 180,E1 -23054.224,E2 -23054.224} C_VEL
LIN {X 0,Y 171.547,Z 421.741,A -85,B 0,C 180,E1 -23059.562,E2 -23059.562} C_VEL
LIN {X 0,Y 171.502,Z 422.079,A -85,B 0,C 180,E1 -23064.192,E2 -23064.192} C_VEL
LIN {X 0,Y 171.877,Z 424.131,A -85,B 0,C 180,E1 -23069.745,E2 -23069.745} C_VEL
LIN {X 0,Y 173.153,Z 427.251,A -85,B 0,C 180,E1 -23070.77,E2 -23070.77} C_VEL
LIN {X 0,Y 175.409,Z 429.801,A -85,B 0,C 180,E1 -23072.234,E2 -23072.234} C_VEL
LIN {X 0,Y 176.085,Z 430.732,A -85,B 0,C 180,E1 -23072.688,E2 -23072.688} C_VEL
LIN {X 0,Y 177.949,Z 434.209,A -85,B 0,C 180,E1 -23073.996,E2 -23073.996} C_VEL
LIN {X 0,Y 179.634,Z 436.414,A -85,B 0,C 180,E1 -23075.035,E2 -23075.035} C_VEL
LIN {X 0,Y 181.793,Z 440.398,A -85,B 0,C 180,E1 -23076.499,E2 -23076.499} C_VEL
LIN {X 0,Y 183.013,Z 442.587,A -85,B 0,C 180,E1 -23077.286,E2 -23077.286} C_VEL
LIN {X 0,Y 185.587,Z 447.575,A -85,B 0,C 180,E1 -23079.019,E2 -23079.019} C_VEL
LIN {X 0,Y 189.557,Z 456.667,A -85,B 0,C 180,E1 -23081.864,E2 -23081.864} C_VEL
LIN {X 0,Y 192.017,Z 464.568,A -85,B 0,C 180,E1 -23084.06,E2 -23084.06} C_VEL
LIN {X 0,Y 193.458,Z 472.304,A -85,B 0,C 180,E1 -23086.009,E2 -23086.009} C_VEL
LIN {X 0,Y 194.535,Z 483.267,A -85,B 0,C 180,E1 -23088.752,E2 -23088.752} C_VEL
LIN {X 0,Y 194.528,Z 493.065,A -85,B 0,C 180,E1 -23091.256,E2 -23091.256} C_VEL
LIN {X 0,Y 194.154,Z 499.51,A -85,B 0,C 180,E1 -23093.02,E2 -23093.02} C_VEL
LIN {X 0,Y 189.664,Z 510.237,A -85,B 0,C 180,E1 -23095.591,E2 -23095.591} C_VEL
LIN {X 0,Y 185.147,Z 519.96,A -85,B 0,C 180,E1 -23098.537,E2 -23098.537} C_VEL
LIN {X 0,Y 181.237,Z 528.027,A -85,B 0,C 180,E1 -23101.638,E2 -23101.638} C_VEL
LIN {X 0,Y 177.292,Z 535.76,A -85,B 0,C 180,E1 -23105.403,E2 -23105.403} C_VEL
LIN {X 0,Y 174.601,Z 541.157,A -85,B 0,C 180,E1 -23108.76,E2 -23108.76} C_VEL
LIN {X 0,Y 172.445,Z 545.593,A -85,B 0,C 180,E1 -23112.202,E2 -23112.202} C_VEL
LIN {X 0,Y 170.746,Z 549.083,A -85,B 0,C 180,E1 -23115.702,E2 -23115.702} C_VEL
LIN {X 0,Y 169.409,Z 552.477,A -85,B 0,C 180,E1 -23120.448,E2 -23120.448} C_VEL
LIN {X 0,Y 168.859,Z 554.483,A -85,B 0,C 180,E1 -23125.225,E2 -23125.225} C_VEL
LIN {X 0,Y 168.872,Z 555.143,A -85,B 0,C 180,E1 -23130,E2 -23130} C_VEL
LIN {X 0,Y 168.859,Z 554.463,A -85,B 0,C 180,E1 -23134.775,E2 -23134.775} C_VEL
LIN {X 0,Y 169.411,Z 552.44,A -85,B 0,C 180,E1 -23139.552,E2 -23139.552} C_VEL
LIN {X 0,Y 170.741,Z 549.026,A -85,B 0,C 180,E1 -23144.298,E2 -23144.298} C_VEL
LIN {X 0,Y 173.133,Z 544.12,A -85,B 0,C 180,E1 -23148.95,E2 -23148.95} C_VEL
LIN {X 0,Y 173.526,Z 543.303,A -85,B 0,C 180,E1 -23149.602,E2 -23149.602} C_VEL
LIN {X 0,Y 174.032,Z 541.01,A -85,B 0,C 180,E1 -23151.391,E2 -23151.391} C_VEL
LIN {X 0,Y 173.4,Z 536.927,A -85,B 0,C 180,E1 -23154.37,E2 -23154.37} C_VEL
LIN {X 0,Y 173.161,Z 532.305,A -85,B 0,C 180,E1 -23157.272,E2 -23157.272} C_VEL
LIN {X 0,Y 174.249,Z 529.161,A -85,B 0,C 180,E1 -23158.882,E2 -23158.882} C_VEL
LIN {X 0,Y 178.434,Z 521.203,A -85,B 0,C 180,E1 -23162.122,E2 -23162.122} C_VEL
LIN {X 0,Y 183.026,Z 511.74,A -85,B 0,C 180,E1 -23165.168,E2 -23165.168} C_VEL
LIN {X 0,Y 187.602,Z 501.591,A -85,B 0,C 180,E1 -23167.735,E2 -23167.735} C_VEL
LIN {X 0,Y 188.174,Z 497.709,A -85,B 0,C 180,E1 -23168.831,E2 -23168.831} C_VEL
LIN {X 0,Y 188.56,Z 486.956,A -85,B 0,C 180,E1 -23171.803,E2 -23171.803} C_VEL
LIN {X 0,Y 187.887,Z 476.009,A -85,B 0,C 180,E1 -23174.708,E2 -23174.708} C_VEL
LIN {X 0,Y 186.674,Z 467.999,A -85,B 0,C 180,E1 -23176.859,E2 -23176.859} C_VEL
LIN {X 0,Y 184.661,Z 460.831,A -85,B 0,C 180,E1 -23178.965,E2 -23178.965} C_VEL
LIN {X 0,Y 180.692,Z 451.073,A -85,B 0,C 180,E1 -23182.223,E2 -23182.223} C_VEL
LIN {X 0,Y 177.83,Z 445.548,A -85,B 0,C 180,E1 -23184.343,E2 -23184.343} C_VEL
LIN {X 0,Y 175.359,Z 440.879,A -85,B 0,C 180,E1 -23186.215,E2 -23186.215} C_VEL
LIN {X 0,Y 173.133,Z 437.165,A -85,B 0,C 180,E1 -23187.874,E2 -23187.874} C_VEL
LIN {X 0,Y 172.403,Z 435.803,A -85,B 0,C 180,E1 -23188.464,E2 -23188.464} C_VEL
LIN {X 0,Y 170.018,Z 432.672,A -85,B 0,C 180,E1 -23190.205,E2 -23190.205} C_VEL
LIN {X 0,Y 168.83,Z 430.082,A -85,B 0,C 180,E1 -23191.262,E2 -23191.262} C_VEL
LIN {X 0,Y 166.351,Z 427.68,A -85,B 0,C 180,E1 -23193.16,E2 -23193.16} C_VEL
LIN {X 0,Y 164.883,Z 424.861,A -85,B 0,C 180,E1 -23194.511,E2 -23194.511} C_VEL
LIN {X 0,Y 164.598,Z 423.832,A -85,B 0,C 180,E1 -23194.893,E2 -23194.893} C_VEL
LIN {X 0,Y 164.485,Z 422.621,A -85,B 0,C 180,E1 -23200.051,E2 -23200.051} C_VEL
LIN {X 0,Y 164.554,Z 422.607,A -85,B 0,C 180,E1 -23205.152,E2 -23205.152} C_VEL
LIN {X 0,Y 164.854,Z 422.572,A -85,B 0,C 180,E1 -23210.182,E2 -23210.182} C_VEL
LIN {X 0,Y 164.864,Z 422.566,A -85,B 0,C 180,E1 -23212.653,E2 -23212.653} C_VEL
LIN {X 0,Y 165.053,Z 422.549,A -85,B 0,C 180,E1 -23217.56,E2 -23217.56} C_VEL
LIN {X 0,Y 165.299,Z 422.518,A -85,B 0,C 180,E1 -23220,E2 -23220} C_VEL
LIN {X 0,Y 164.864,Z 422.575,A -85,B 0,C 180,E1 -23227.348,E2 -23227.348} C_VEL
LIN {X 0,Y 164.781,Z 422.584,A -85,B 0,C 180,E1 -23231.198,E2 -23231.198} C_VEL
LIN {X 0,Y 164.506,Z 422.612,A -85,B 0,C 180,E1 -23237.401,E2 -23237.401} C_VEL
LIN {X 0,Y 164.474,Z 422.622,A -85,B 0,C 180,E1 -23239.989,E2 -23239.989} C_VEL
LIN {X 0,Y 164.447,Z 422.818,A -85,B 0,C 180,E1 -23245.132,E2 -23245.132} C_VEL
LIN {X 0,Y 165.382,Z 425.448,A -85,B 0,C 180,E1 -23246.122,E2 -23246.122} C_VEL
LIN {X 0,Y 167.705,Z 428.068,A -85,B 0,C 180,E1 -23248.01,E2 -23248.01} C_VEL
LIN {X 0,Y 168.89,Z 428.946,A -85,B 0,C 180,E1 -23248.88,E2 -23248.88} C_VEL
LIN {X 0,Y 170.712,Z 432.502,A -85,B 0,C 180,E1 -23250.435,E2 -23250.435} C_VEL
LIN {X 0,Y 172.771,Z 435.033,A -85,B 0,C 180,E1 -23251.926,E2 -23251.926} C_VEL
LIN {X 0,Y 174.85,Z 438.694,A -85,B 0,C 180,E1 -23253.537,E2 -23253.537} C_VEL
LIN {X 0,Y 175.902,Z 440.237,A -85,B 0,C 180,E1 -23254.271,E2 -23254.271} C_VEL
LIN {X 0,Y 178.884,Z 445.922,A -85,B 0,C 180,E1 -23256.546,E2 -23256.546} C_VEL
LIN {X 0,Y 181.944,Z 452.135,A -85,B 0,C 180,E1 -23258.881,E2 -23258.881} C_VEL
LIN {X 0,Y 185.549,Z 461.387,A -85,B 0,C 180,E1 -23261.969,E2 -23261.969} C_VEL
LIN {X 0,Y 187.575,Z 469.343,A -85,B 0,C 180,E1 -23264.317,E2 -23264.317} C_VEL
LIN {X 0,Y 188.87,Z 478.486,A -85,B 0,C 180,E1 -23266.844,E2 -23266.844} C_VEL
LIN {X 0,Y 189.328,Z 487.678,A -85,B 0,C 180,E1 -23269.4,E2 -23269.4} C_VEL
LIN {X 0,Y 189.046,Z 495.502,A -85,B 0,C 180,E1 -23271.634,E2 -23271.634} C_VEL
LIN {X 0,Y 188.1,Z 498.47,A -85,B 0,C 180,E1 -23272.352,E2 -23272.352} C_VEL
LIN {X 0,Y 183.48,Z 508.713,A -85,B 0,C 180,E1 -23274.931,E2 -23274.931} C_VEL
LIN {X 0,Y 178.934,Z 518.165,A -85,B 0,C 180,E1 -23277.979,E2 -23277.979} C_VEL
LIN {X 0,Y 174.188,Z 527.177,A -85,B 0,C 180,E1 -23281.701,E2 -23281.701} C_VEL
LIN {X 0,Y 170.326,Z 534.437,A -85,B 0,C 180,E1 -23285.631,E2 -23285.631} C_VEL
LIN {X 0,Y 167.634,Z 539.519,A -85,B 0,C 180,E1 -23289.123,E2 -23289.123} C_VEL
LIN {X 0,Y 164.71,Z 544.782,A -85,B 0,C 180,E1 -23293.898,E2 -23293.898} C_VEL
LIN {X 0,Y 163.287,Z 547.72,A -85,B 0,C 180,E1 -23297.573,E2 -23297.573} C_VEL
LIN {X 0,Y 162.198,Z 550.414,A -85,B 0,C 180,E1 -23302.531,E2 -23302.531} C_VEL
LIN {X 0,Y 161.762,Z 551.797,A -85,B 0,C 180,E1 -23307.818,E2 -23307.818} C_VEL
LIN {X 0,Y 161.765,Z 551.806,A -85,B 0,C 180,E1 -23312.21,E2 -23312.21} C_VEL
LIN {X 0,Y 162.194,Z 550.483,A -85,B 0,C 180,E1 -23317.469,E2 -23317.469} C_VEL
LIN {X 0,Y 163.266,Z 547.831,A -85,B 0,C 180,E1 -23322.429,E2 -23322.429} C_VEL
LIN {X 0,Y 165.257,Z 543.755,A -85,B 0,C 180,E1 -23327.319,E2 -23327.319} C_VEL
LIN {X 0,Y 168.425,Z 538.122,A -85,B 0,C 180,E1 -23332.059,E2 -23332.059} C_VEL
LIN {X 0,Y 171.543,Z 532.286,A -85,B 0,C 180,E1 -23335.791,E2 -23335.791} C_VEL
LIN {X 0,Y 175.414,Z 525.083,A -85,B 0,C 180,E1 -23339.393,E2 -23339.393} C_VEL
LIN {X 0,Y 179.578,Z 517.062,A -85,B 0,C 180,E1 -23342.556,E2 -23342.556} C_VEL
LIN {X 0,Y 184.294,Z 507.387,A -85,B 0,C 180,E1 -23345.56,E2 -23345.56} C_VEL
LIN {X 0,Y 188.75,Z 497.118,A -85,B 0,C 180,E1 -23348.096,E2 -23348.096} C_VEL
LIN {X 0,Y 189.152,Z 494.876,A -85,B 0,C 180,E1 -23348.715,E2 -23348.715} C_VEL
LIN {X 0,Y 189.363,Z 485.339,A -85,B 0,C 180,E1 -23351.411,E2 -23351.411} C_VEL
LIN {X 0,Y 188.717,Z 475.99,A -85,B 0,C 180,E1 -23353.988,E2 -23353.988} C_VEL
LIN {X 0,Y 187.229,Z 467.263,A -85,B 0,C 180,E1 -23356.444,E2 -23356.444} C_VEL
LIN {X 0,Y 184.766,Z 458.981,A -85,B 0,C 180,E1 -23358.993,E2 -23358.993} C_VEL
LIN {X 0,Y 181.442,Z 451.152,A -85,B 0,C 180,E1 -23361.702,E2 -23361.702} C_VEL
LIN {X 0,Y 177.8,Z 443.736,A -85,B 0,C 180,E1 -23364.51,E2 -23364.51} C_VEL
LIN {X 0,Y 175.318,Z 439.215,A -85,B 0,C 180,E1 -23366.399,E2 -23366.399} C_VEL
LIN {X 0,Y 173.084,Z 435.744,A -85,B 0,C 180,E1 -23368.053,E2 -23368.053} C_VEL
LIN {X 0,Y 172.495,Z 434.344,A -85,B 0,C 180,E1 -23368.583,E2 -23368.583} C_VEL
LIN {X 0,Y 169.965,Z 431.34,A -85,B 0,C 180,E1 -23370.421,E2 -23370.421} C_VEL
LIN {X 0,Y 168.705,Z 428.729,A -85,B 0,C 180,E1 -23371.545,E2 -23371.545} C_VEL
LIN {X 0,Y 165.948,Z 426.243,A -85,B 0,C 180,E1 -23373.691,E2 -23373.691} C_VEL
LIN {X 0,Y 164.665,Z 423.801,A -85,B 0,C 180,E1 -23374.904,E2 -23374.904} C_VEL
LIN {X 0,Y 164.426,Z 422.626,A -85,B 0,C 180,E1 -23375.287,E2 -23375.287} C_VEL
LIN {X 0,Y 164.487,Z 422.614,A -85,B 0,C 180,E1 -23380.051,E2 -23380.051} C_VEL
LIN {X 0,Y 164.539,Z 422.614,A -85,B 0,C 180,E1 -23385.15,E2 -23385.15} C_VEL
LIN {X 0,Y 164.856,Z 422.576,A -85,B 0,C 180,E1 -23390.181,E2 -23390.181} C_VEL
LIN {X 0,Y 164.865,Z 422.574,A -85,B 0,C 180,E1 -23392.652,E2 -23392.652} C_VEL
LIN {X 0,Y 165.053,Z 422.551,A -85,B 0,C 180,E1 -23397.559,E2 -23397.559} C_VEL
LIN {X 0,Y 165.298,Z 422.52,A -85,B 0,C 180,E1 -23400,E2 -23400} C_VEL
LIN {X 0,Y 164.779,Z 422.584,A -85,B 0,C 180,E1 -23404.893,E2 -23404.893} C_VEL
LIN {X 0,Y 164.865,Z 422.573,A -85,B 0,C 180,E1 -23407.347,E2 -23407.347} C_VEL
LIN {X 0,Y 164.782,Z 422.585,A -85,B 0,C 180,E1 -23411.198,E2 -23411.198} C_VEL
LIN {X 0,Y 164.508,Z 422.617,A -85,B 0,C 180,E1 -23417.4,E2 -23417.4} C_VEL
LIN {X 0,Y 164.475,Z 422.623,A -85,B 0,C 180,E1 -23419.989,E2 -23419.989} C_VEL
LIN {X 0,Y 164.621,Z 423.838,A -85,B 0,C 180,E1 -23424.934,E2 -23424.934} C_VEL
LIN {X 0,Y 165.89,Z 426.954,A -85,B 0,C 180,E1 -23426.232,E2 -23426.232} C_VEL
LIN {X 0,Y 168.326,Z 429.728,A -85,B 0,C 180,E1 -23428.185,E2 -23428.185} C_VEL
LIN {X 0,Y 169.143,Z 430.488,A -85,B 0,C 180,E1 -23428.798,E2 -23428.798} C_VEL
LIN {X 0,Y 170.904,Z 434.055,A -85,B 0,C 180,E1 -23430.31,E2 -23430.31} C_VEL
LIN {X 0,Y 172.871,Z 436.437,A -85,B 0,C 180,E1 -23431.716,E2 -23431.716} C_VEL
LIN {X 0,Y 174.947,Z 440.352,A -85,B 0,C 180,E1 -23433.357,E2 -23433.357} C_VEL
LIN {X 0,Y 176.098,Z 442.033,A -85,B 0,C 180,E1 -23434.154,E2 -23434.154} C_VEL
LIN {X 0,Y 178.372,Z 446.307,A -85,B 0,C 180,E1 -23435.88,E2 -23435.88} C_VEL
LIN {X 0,Y 182.188,Z 454.411,A -85,B 0,C 180,E1 -23438.819,E2 -23438.819} C_VEL
LIN {X 0,Y 185.373,Z 462.866,A -85,B 0,C 180,E1 -23441.565,E2 -23441.565} C_VEL
LIN {X 0,Y 187.13,Z 469.869,A -85,B 0,C 180,E1 -23443.592,E2 -23443.592} C_VEL
LIN {X 0,Y 188.405,Z 480.434,A -85,B 0,C 180,E1 -23446.392,E2 -23446.392} C_VEL
LIN {X 0,Y 188.658,Z 490.385,A -85,B 0,C 180,E1 -23449.074,E2 -23449.074} C_VEL
LIN {X 0,Y 187.98,Z 500.568,A -85,B 0,C 180,E1 -23451.948,E2 -23451.948} C_VEL
LIN {X 0,Y 183.836,Z 510.171,A -85,B 0,C 180,E1 -23454.337,E2 -23454.337} C_VEL
LIN {X 0,Y 179.102,Z 519.893,A -85,B 0,C 180,E1 -23457.346,E2 -23457.346} C_VEL
LIN {X 0,Y 174.98,Z 527.959,A -85,B 0,C 180,E1 -23460.526,E2 -23460.526} C_VEL
LIN {X 0,Y 170.827,Z 535.692,A -85,B 0,C 180,E1 -23464.406,E2 -23464.406} C_VEL
LIN {X 0,Y 167.959,Z 541.089,A -85,B 0,C 180,E1 -23467.877,E2 -23467.877} C_VEL
LIN {X 0,Y 165.651,Z 545.525,A -85,B 0,C 180,E1 -23471.446,E2 -23471.446} C_VEL
LIN {X 0,Y 163.822,Z 549.014,A -85,B 0,C 180,E1 -23475.084,E2 -23475.084} C_VEL
LIN {X 0,Y 162.389,Z 552.409,A -85,B 0,C 180,E1 -23480.031,E2 -23480.031} C_VEL
LIN {X 0,Y 161.766,Z 554.414,A -85,B 0,C 180,E1 -23485.015,E2 -23485.015} C_VEL
LIN {X 0,Y 161.772,Z 555.074,A -85,B 0,C 180,E1 -23490,E2 -23490} C_VEL
LIN {X 0,Y 161.766,Z 554.394,A -85,B 0,C 180,E1 -23494.985,E2 -23494.985} C_VEL
LIN {X 0,Y 162.39,Z 552.371,A -85,B 0,C 180,E1 -23499.969,E2 -23499.969} C_VEL
LIN {X 0,Y 163.818,Z 548.956,A -85,B 0,C 180,E1 -23504.916,E2 -23504.916} C_VEL
LIN {X 0,Y 166.402,Z 544.049,A -85,B 0,C 180,E1 -23509.748,E2 -23509.748} C_VEL
LIN {X 0,Y 169.606,Z 537.795,A -85,B 0,C 180,E1 -23514.27,E2 -23514.27} C_VEL
LIN {X 0,Y 173.676,Z 530.223,A -85,B 0,C 180,E1 -23518.39,E2 -23518.39} C_VEL
LIN {X 0,Y 174.249,Z 529.161,A -85,B 0,C 180,E1 -23518.882,E2 -23518.882} C_VEL
LIN {X 0,Y 175.446,Z 525.862,A -85,B 0,C 180,E1 -23520.44,E2 -23520.44} C_VEL
LIN {X 0,Y 175.917,Z 520.24,A -85,B 0,C 180,E1 -23523.1,E2 -23523.1} C_VEL
LIN {X 0,Y 176.578,Z 514.151,A -85,B 0,C 180,E1 -23525.629,E2 -23525.629} C_VEL
LIN {X 0,Y 178.015,Z 510.091,A -85,B 0,C 180,E1 -23526.936,E2 -23526.936} C_VEL
LIN {X 0,Y 181.507,Z 502.706,A -85,B 0,C 180,E1 -23528.837,E2 -23528.837} C_VEL
LIN {X 0,Y 182.201,Z 497.541,A -85,B 0,C 180,E1 -23530.389,E2 -23530.389} C_VEL
LIN {X 0,Y 182.659,Z 487.188,A -85,B 0,C 180,E1 -23533.389,E2 -23533.389} C_VEL
LIN {X 0,Y 182.109,Z 476.533,A -85,B 0,C 180,E1 -23536.383,E2 -23536.383} C_VEL
LIN {X 0,Y 180.799,Z 468.973,A -85,B 0,C 180,E1 -23538.638,E2 -23538.638} C_VEL
LIN {X 0,Y 178.654,Z 461.912,A -85,B 0,C 180,E1 -23540.993,E2 -23540.993} C_VEL
LIN {X 0,Y 175.56,Z 454.343,A -85,B 0,C 180,E1 -23543.81,E2 -23543.81} C_VEL
LIN {X 0,Y 173.612,Z 450.285,A -85,B 0,C 180,E1 -23545.477,E2 -23545.477} C_VEL
LIN {X 0,Y 171.678,Z 446.342,A -85,B 0,C 180,E1 -23547.152,E2 -23547.152} C_VEL
LIN {X 0,Y 169.541,Z 442.175,A -85,B 0,C 180,E1 -23549.051,E2 -23549.051} C_VEL
LIN {X 0,Y 166.869,Z 438.175,A -85,B 0,C 180,E1 -23551.286,E2 -23551.286} C_VEL
LIN {X 0,Y 166.15,Z 436.347,A -85,B 0,C 180,E1 -23552.058,E2 -23552.058} C_VEL
LIN {X 0,Y 163.726,Z 433.672,A -85,B 0,C 180,E1 -23554.132,E2 -23554.132} C_VEL
LIN {X 0,Y 161.996,Z 430.132,A -85,B 0,C 180,E1 -23556,E2 -23556} C_VEL
LIN {X 0,Y 159.037,Z 427.45,A -85,B 0,C 180,E1 -23558.958,E2 -23558.958} C_VEL
LIN {X 0,Y 157.529,Z 424.179,A -85,B 0,C 180,E1 -23560.947,E2 -23560.947} C_VEL
LIN {X 0,Y 157.44,Z 423.647,A -85,B 0,C 180,E1 -23561.222,E2 -23561.222} C_VEL
LIN {X 0,Y 157.56,Z 423.484,A -85,B 0,C 180,E1 -23567.113,E2 -23567.113} C_VEL
LIN {X 0,Y 157.773,Z 423.451,A -85,B 0,C 180,E1 -23569.736,E2 -23569.736} C_VEL
LIN {X 0,Y 157.826,Z 423.443,A -85,B 0,C 180,E1 -23572.323,E2 -23572.323} C_VEL
LIN {X 0,Y 158.261,Z 423.395,A -85,B 0,C 180,E1 -23580,E2 -23580} C_VEL
LIN {X 0,Y 157.826,Z 423.452,A -85,B 0,C 180,E1 -23587.677,E2 -23587.677} C_VEL
LIN {X 0,Y 157.707,Z 423.466,A -85,B 0,C 180,E1 -23591.363,E2 -23591.363} C_VEL
LIN {X 0,Y 157.479,Z 423.495,A -85,B 0,C 180,E1 -23595.532,E2 -23595.532} C_VEL
LIN {X 0,Y 157.438,Z 423.56,A -85,B 0,C 180,E1 -23599.063,E2 -23599.063} C_VEL
LIN {X 0,Y 158.157,Z 425.84,A -85,B 0,C 180,E1 -23600.162,E2 -23600.162} C_VEL
LIN {X 0,Y 159.574,Z 427.849,A -85,B 0,C 180,E1 -23601.815,E2 -23601.815} C_VEL
LIN {X 0,Y 162.115,Z 429.604,A -85,B 0,C 180,E1 -23604.265,E2 -23604.265} C_VEL
LIN {X 0,Y 163.473,Z 432.461,A -85,B 0,C 180,E1 -23605.756,E2 -23605.756} C_VEL
LIN {X 0,Y 166.174,Z 435.401,A -85,B 0,C 180,E1 -23608.102,E2 -23608.102} C_VEL
LIN {X 0,Y 168.205,Z 439.134,A -85,B 0,C 180,E1 -23609.999,E2 -23609.999} C_VEL
LIN {X 0,Y 169.51,Z 440.853,A -85,B 0,C 180,E1 -23611.042,E2 -23611.042} C_VEL
LIN {X 0,Y 171.587,Z 444.66,A -85,B 0,C 180,E1 -23612.868,E2 -23612.868} C_VEL
LIN {X 0,Y 174.824,Z 451.037,A -85,B 0,C 180,E1 -23615.656,E2 -23615.656} C_VEL
LIN {X 0,Y 178.6,Z 459.688,A -85,B 0,C 180,E1 -23619.022,E2 -23619.022} C_VEL
LIN {X 0,Y 181.072,Z 467.484,A -85,B 0,C 180,E1 -23621.704,E2 -23621.704} C_VEL
LIN {X 0,Y 182.442,Z 474.596,A -85,B 0,C 180,E1 -23623.9,E2 -23623.9} C_VEL
LIN {X 0,Y 183.238,Z 482.891,A -85,B 0,C 180,E1 -23626.34,E2 -23626.34} C_VEL
LIN {X 0,Y 183.248,Z 492.841,A -85,B 0,C 180,E1 -23629.308,E2 -23629.308} C_VEL
LIN {X 0,Y 182.818,Z 497.823,A -85,B 0,C 180,E1 -23630.825,E2 -23630.825} C_VEL
LIN {X 0,Y 177.706,Z 508.785,A -85,B 0,C 180,E1 -23633.614,E2 -23633.614} C_VEL
